(* CODESYS project cnc_v3.project
   Version: 0.0.0.0
   Title: cnc
   Author: Officina

Project tree, tasks and I/O mapping:
  MyController : TM241C24R, Schneider Electric, order no. TM241C24R, version 5.0.8.2
    application Application
      libraries: SysTimeCore, * (System); MemoryUtils, * (3S - Smart Software Solutions GmbH); CAA Mathematics, * (CAA Technical Workgroup); FloatingPointUtils, * (System); VisuDialogs, * (System)
      task MAST (cyclic, interval 20 ms, priority 15, watchdog 100 ms x 1) calls test
      program test [CFC]
      cnc/
        function block cnc [ST]: line_lenght, sc_char_is_letter, sc_findp, sc_find_nonum, sc_find_num, sc_get_letter, sc_get_value, sc_parse_clean, sc_parse_line, sc_parse_start, to_upper, trim, uppercase, arc_lenght, line_arc_angle, arc_arc_angle, line_line_angle, arc_line_angle, p_to_v, get_blockangles, get_corner_ve_blockangles, sc_get_gforce, get_velmax_gforce, sc_optimize_all, sc_optimize_G0_ve, sc_optimize_G123_ve_backward, sc_optimize_G123_ve_forward, sc_set_gforce, interpolate_lenght, interpolate_arc, update_motion_and_interpolator, interpolate_line, round, netto, set_pnt_at
        structure/
          data type sc_motion_status
          data type sc_data
          data type sc_enum_program_status
          data type sc_segment
          data type coordinate_type
          data type sc_pnt
          data type sc_primitive_id
          data type ascii_letters
          data type sc_dir
          data type sc_ext
          data type cn_jog_cmd
          data type cn_limits
        vector3/
          function V3_ANG [ST]
          function V3_DOT [ST]
          function V3_NORMALIZED [ST]
          function V3_NUL [ST]
          function V3_PAR [ST]
          function V3_REV [ST]
          function V3_SMUL [ST]
          function V3_SUB [ST]
          function V3_XANG [ST]
          function V3_CROSS [ST]
          function V3_YANG [ST]
          function V3_ZANG [ST]
          function V3_COPY [ST]
          function V3_NORM [ST]
          function V3_SDIV [ST]
          data type Vector_3
          function V3_ABS [ST]
          function V3_ADD [ST]
        motion/
          function block sc_engine [ST]: set_data, get_result, set_cycle_time, update, motion, Sc_bck, Sc_fwd, get_status, set_pos, set_jog, jog_stop
        global variables CN_CONSTANT
        vector/
          functions/
            function vector_traject_lenght [ST]
            function vector_nr_decrement [ST]
            function vector_at [ST]
            function vector_nr_increment [ST]
            function round [ST]
          function block vector_sc_segment [ST]: clear, end, begin, push_back, back, front, size, insert
        global variables CN_SETTINGS
      trace Traccia (task MAST): test.x, test.y, test.z, test.velocity, test.acceleration
      visualisation Visualization
      new/
        function block sc_parser [ST]: arc_lenght, line_lenght, sc_char_is_letter, sc_findp, sc_find_nonum, sc_find_num, sc_get_letter, sc_get_value, sc_parse_clean, sc_parse_line, sc_parse_start, to_upper, trim, uppercase
        function block sc_optimizer [ST]: arc_arc_angle, arc_line_angle, get_blockangles, get_corner_ve_blockangles, get_velmax_gforce, line_arc_angle, line_line_angle, p_to_v, sc_get_gforce, sc_optimize_all, sc_optimize_G0_ve, sc_optimize_G123_ve_backward, sc_optimize_G123_ve_forward, sc_set_gforce
    Serial_Line_2 : Serial line, Schneider Electric, version 5.0.8.2
      Modbus_Manager : Modbus Manager, Schneider Electric, version 4.0.0.3
    DI : Digital Inputs, Schneider Electric, version 5.0.8.2
        input  iwDI_IW0 : WORD  // IW0
        input  ibDI_IB1 : BYTE  // IB1
    DQ : Digital Outputs, Schneider Electric, version 5.0.8.2
        output qwDQ_QW0 : WORD  // QW0
        output qbDQ_QB1 : BYTE  // QB1
    Counters : Counters, Schneider Electric, version 5.0.8.2
    Pulse_Generators : Pulse Generators, Schneider Electric, version 5.0.8.2
    IO_Bus : IO bus - TM3, Schneider Electric, version 5.0.8.2
    Serial_Line_1 : Serial line, Schneider Electric, version 5.0.8.2
      Machine_Expert_Network_Manager : Machine Expert-Network Manager, Schneider Electric, version 4.0.0.3
    Cartridge_1 : Cartridge, Schneider Electric, version 5.0.8.2
    COM_Bus : COM bus, Schneider Electric, version 5.0.8.2
  libraries: VisuSymbols, 3.5.10.0 (System)
  text list GlobalTextList
*)

// MyController/Application/cnc/structure/sc_motion_status
TYPE sc_motion_status :
(
	motion_error,
	motion_finish,
	motion_pause,
	motion_process
);
END_TYPE

// MyController/Application/cnc/structure/sc_data
TYPE sc_data :
STRUCT
	sc_ct:LREAL;//scurve curve time                 //
	sc_jm:LREAL;//jerk result                       //
 	sc_cs:LREAL;//curve displacement                //
	sc_vr:LREAL;//velocity resul                    //
	sc_sr:LREAL;//position result                   //  result
	sc_ar:LREAL;//acceleration result               //
	tr_ct:LREAL;//total curve time                  //
 	tr_cs:LREAL;//total curve displacement          //
	at_time:LREAL;//request at timestamp.			//
	cycle_time:LREAL;
	state:sc_motion_status;
	
	ds:LREAL;//target
	vo:LREAL;//begin velocity
	ve:LREAL;//end velocity
	vs:LREAL;//max velocity
	a:LREAL;//acceleration
	gain:LREAL;//0-100
	
	ds_old:LREAL;//target old
	vs_old:LREAL;//max velocity old
	sc_sr_inc:LREAL;//position result incremental
	sc_sr_inc_old:LREAL;//position result incremental old
		
	init:BOOL;//new move reinit
	stop:BOOL;
	zero_vel_acc:BOOL;
	
	dir:INT;//movement direction
	
	t_vin:LREAL;
	t_pos:LREAL;
	
	finish:BOOL;
	
	jog_stop:BOOL;
	jog_fwd:BOOL;
	jog_rev:BOOL;
	
END_STRUCT
END_TYPE

// MyController/Application/cnc/structure/sc_enum_program_status

TYPE sc_enum_program_status :
(
	program_start:=0,
	program_run:=1,
	program_pause:=2,
	program_pause_resume:=3,
	program_stop:=4,
	program_vm_interupt:=5,
	program_wait:=6,
	program_end:=7,
	program_jog:=8,
	program_error:=9
);
END_TYPE

// MyController/Application/cnc/structure/sc_segment
TYPE sc_segment :
STRUCT
	primitive_id:sc_primitive_id;
    gcode_line_nr:UDINT;
    pnt_s:sc_pnt; 
	pnt_e:sc_pnt;
	pnt_c:sc_pnt;
   	dir_s:sc_dir; 
	dir_e:sc_dir;
    ext_s:sc_ext; 
	ext_e:sc_ext;
	radius:LREAL;
    angle_end:LREAL;
	vel_start:LREAL;
	vel_max:LREAL;
    vel_end:LREAL;
	acc_start:LREAL;
	acc_end:LREAL;
    traject_lenght_begin:LREAL;
	traject_lenght_end:LREAL;
    path_lenght:LREAL;
	m_value:UDINT;
	s_value:UDINT;
	s_dir:BOOL; //! spindle direction (1cw -0ccw)
	p_value:UDINT;
	t_value:UDINT;
	h_value:UDINT;
	abs_inc:BOOL;//abs / inc coordinate 
	back_optim:BOOL;
	forward_optim:BOOL;
END_STRUCT
END_TYPE

// MyController/Application/cnc/structure/coordinate_type

TYPE coordinate_type :
(
	abs_coord := 0,
	inc_coord := 1
);
END_TYPE

// MyController/Application/cnc/structure/sc_pnt
TYPE sc_pnt :
STRUCT
	x,y,z:LREAL;
END_STRUCT
END_TYPE

// MyController/Application/cnc/structure/sc_primitive_id

TYPE sc_primitive_id :
(
	empty:=0,
	rapid:=1,
	line:=2,
	arc_cw:=3,
	arc_ccw:=4	
);
END_TYPE

// MyController/Application/cnc/structure/ascii_letters

TYPE ascii_letters :
(
        A_ := 65,
        B_ := 66,
        C_ := 67,
        D_ := 68,
        E_ := 69,
        F_ := 70,
        G_ := 71,
        H_ := 72,
        I_ := 73,
        J_ := 74,
        K_ := 75,
        L_ := 76,
        M_ := 77,
        N_ := 78,
        O_ := 79,
        P_ := 80,
        Q_ := 81,
        R_ := 82,
        S_ := 83,
        T_ := 84,
        U_ := 85,
        V_ := 86,
        W_ := 87,
        X_ := 88,
        Y_ := 89,
        Z_ := 90
);
END_TYPE

// MyController/Application/cnc/structure/sc_dir
TYPE sc_dir :
STRUCT
	a:LREAL;
	b:LREAL;
	c:LREAL;
END_STRUCT
END_TYPE

// MyController/Application/cnc/structure/sc_ext
TYPE sc_ext :
STRUCT
	u:LREAL;
	v:LREAL;
	w:LREAL;
END_STRUCT
END_TYPE

// MyController/Application/cnc/vector3/Vector_3
TYPE Vector_3 :
STRUCT
	x:LREAL;
	y:LREAL;
	z:LREAL;
END_STRUCT
END_TYPE

// MyController/Application/cnc/structure/cn_jog_cmd
TYPE cn_jog_cmd :
STRUCT
	jog_enable:BOOL;
	x_up:BOOL;
	x_dn:BOOL;
	y_up:BOOL;
	y_dn:BOOL;
	z_up:BOOL;
	z_dp:BOOL;
END_STRUCT
END_TYPE

// MyController/Application/cnc/structure/cn_limits
TYPE cn_limits :
STRUCT
	max_vel:LREAL;
	max_acc:LREAL;
	max_jerk:LREAL;
	max_quote_x:LREAL;
	min_quote_x:LREAL;
	max_quote_y:LREAL;
	min_quote_y:LREAL;
	max_quote_z:LREAL;
	min_quote_z:LREAL;
END_STRUCT
END_TYPE

// MyController/Application/cnc/CN_CONSTANT
VAR_GLOBAL CONSTANT	
	DECIMALS:INT:=3;
	INFINITY:LREAL:=3.402823E+38;			
	M_PI:LREAL:=3.14159265358979323846264338327950288;
	TO_DEGREES:LREAL:=180/M_PI;
END_VAR

// MyController/Application/cnc/CN_SETTINGS
VAR_GLOBAL CONSTANT
	ANGLE_VEL_FACTOR:LREAL:=1;// 0-1
	STOP_ANGLE:LREAL:=90; 
	CT:LREAL:=0.02; //cycle time
	MAX_LOOK_HEAD_LINE:UDINT:=50;
	MAX_GCODE_LINE:UDINT:=2500;
	MAX_TOOLS:UINT:=10;
END_VAR

// MyController/Application/test
PROGRAM test
VAR
	cnc_0: cnc;
	feed_override: LREAL:=100;
	adaptive_feed: LREAL:=100;
	maxacc: LREAL:=250;
	maxjerk: LREAL:=100;
	maxvel: LREAL:=250;
	start: BOOL;
	stop: BOOL;
	pause: BOOL;
	start_line: UDINT;
	x: LREAL;
	y: LREAL;
	z: LREAL;
	velocity: LREAL;
	acceleration: LREAL;
	traject_progress: LREAL;
	line_progress: LREAL;
	performance: LREAL;
	line_nr: UDINT;
	jog_enable: BOOL;
	gcode:ARRAY [0..MAX_GCODE_LINE]OF STRING (250)
	:=[		
		
'G1 X0 Y50 z0 F150 						',			
'G1 X10 Y100 z0							',
'G1 X0 Y150 z0 							',
'G2 X150 Y0 z-15 I0 J-150 				',
'G0 z2                          ',
'G00 X-25.967 Y-14.626 Z2.000   ',
'G00 X0.033 Y0.040 Z2.000       ',
'G01 X0.033 Y0.040 Z-0.160 F50 ',
'G01 X-0.078 Y-0.152 Z-0.160    ',
'G01 X-0.189 Y0.425 Z-0.242     ',
'G01 X0.700 Y0.040 Z-0.019      ',
'G01 X0.601 Y-0.436 Z-0.019     ',
'G01 X0.175 Y-0.762 Z-0.097     ',
'G01 X-0.411 Y-0.729 Z-0.343    ',
'G01 X-0.872 Y-0.289 Z-0.610    ',
'G01 X-0.941 Y0.395 Z-0.610     ',
'G01 X-0.522 Y1.003 Z-0.347     ',
'G01 X0.239 Y1.208 Z-0.102      ',
'G01 X0.998 Y0.850 Z-0.005      ',
'G01 X1.367 Y0.040 Z0.000       ',
'G01 X1.292 Y-0.520 Z0.000      ',
'G01 X0.985 Y-1.016 Z-0.006     ',
'G01 X0.487 Y-1.354 Z-0.058     ',
'G01 X-0.125 Y-1.462 Z-0.267    ',
'G01 X-0.744 Y-1.307 Z-0.486    ',
'G01 X-1.261 Y-0.900 Z-0.937    ',
'G01 X-1.575 Y-0.301 Z-1.036    ',
'G01 X-1.619 Y0.392 Z-1.036     ',
'G01 X-1.369 Y1.059 Z-0.951     ',
'G01 X-0.856 Y1.580 Z-0.660     ',
'G01 X-0.157 Y1.853 Z-0.288     ',
'G01 X0.610 Y1.816 Z-0.035      ',
'G01 X1.312 Y1.461 Z0.000       ',
'G01 X1.820 Y0.836 Z0.000       ',
'G01 X2.033 Y0.040 Z0.000       ',
'G01 X1.975 Y-0.558 Z0.000      ',
'G01 X1.738 Y-1.122 Z0.000      ',
'G01 X1.340 Y-1.598 Z0.000      ',
'G01 X0.810 Y-1.939 Z-0.038     ',
'G01 X0.195 Y-2.112 Z-0.151     ',
'G01 X-0.454 Y-2.095 Z-0.437    ',
'G01 X-1.078 Y-1.884 Z-0.881    ',
'G01 X-1.619 Y-1.493 Z-1.085    ',
'G01 X-2.026 Y-0.951 Z-1.114    ',
'G01 X-2.258 Y-0.305 Z-1.114    ',
'G01 X-2.290 Y0.391 Z-1.114     ',
'G01 X-2.112 Y1.074 Z-1.117     ',
'G01 X-1.735 Y1.682 Z-1.134     ',
'G01 X-1.189 Y2.157 Z-0.927     ',
'G01 X-0.518 Y2.455 Z-0.478     ',
'G01 X0.221 Y2.541 Z-0.174      ',
'G01 X0.961 Y2.405 Z-0.028      ',
'G01 X1.637 Y2.051 Z0.000       ',
'G01 X2.184 Y1.507 Z0.000       ',
'G01 X2.551 Y0.817 Z0.000       ',
'G01 X2.700 Y0.040 Z0.000       ',
'G01 X2.656 Y-0.558 Z0.000      ',
'G01 X2.479 Y-1.137 Z0.000      ',
'G01 X2.174 Y-1.667 Z0.000      ',
'G01 X1.755 Y-2.119 Z0.000      ',
'G01 X1.242 Y-2.469 Z-0.007     ',
'G01 X0.659 Y-2.699 Z-0.071     ',
'G01 X0.033 Y-2.793 Z-0.303     ',
'G01 X-0.602 Y-2.745 Z-0.691    ',
'G01 X-1.217 Y-2.555 Z-1.150    ',
'G01 X-1.778 Y-2.231 Z-1.189    ',
'G01 X-2.256 Y-1.785 Z-1.144    ',
'G01 X-2.627 Y-1.241 Z-1.131    ',
'G01 X-2.868 Y-0.622 Z-1.120    ',
'G01 X-2.967 Y0.040 Z-1.119     ',
'G01 X-2.915 Y0.713 Z-1.120     ',
'G01 X-2.712 Y1.363 Z-1.134     ',
'G01 X-2.368 Y1.955 Z-1.175     ',
'G01 X-1.897 Y2.460 Z-1.230     ',
'G01 X-1.320 Y2.851 Z-1.221     ',
'G01 X-0.666 Y3.105 Z-0.765     ',
'G01 X0.033 Y3.207 Z-0.352      ',
'G01 X0.743 Y3.151 Z-0.112      ',
'G01 X1.428 Y2.936 Z-0.006      ',
'G01 X2.052 Y2.572 Z0.000       ',
'G01 X2.584 Y2.074 Z0.000       ',
'G00 X120 Y120 Z0.000       ',
'G01 X2.994 Y1.466 Z0.000       ',
'G01 X3.260 Y0.777 Z-0.008      ',
'G01 X3.367 Y0.040 Z-0.015      ',
'G01 X3.329 Y-0.576 Z-0.009     ',
'G01 X3.178 Y-1.178 Z0.000      ',
'G01 X2.917 Y-1.745 Z0.000      ',
'G01 X2.555 Y-2.258 Z0.000      ',
'G01 X2.101 Y-2.698 Z0.000      ',
'G01 X1.572 Y-3.049 Z0.000      ',
'G01 X0.983 Y-3.298 Z-0.077     ',
'G01 X0.355 Y-3.435 Z-0.317     ',
'G01 X-0.291 Y-3.454 Z-0.548    ',
'G01 X-0.933 Y-3.354 Z-0.977    ',
'G01 X-1.549 Y-3.136 Z-1.340    ',
'G01 X-2.117 Y-2.807 Z-1.291    ',
'G01 X-2.618 Y-2.377 Z-1.228    ',
'G01 X-3.034 Y-1.859 Z-1.205    ',
'G01 X-3.349 Y-1.270 Z-1.167    ',
'G01 X-3.552 Y-0.630 Z-1.156    ',
'G01 X-3.633 Y0.040 Z-1.156     ',
'G01 X-3.590 Y0.718 Z-1.157     ',
'G01 X-3.422 Y1.379 Z-1.193     ',
'G01 X-3.134 Y2.002 Z-1.212     ',
'G01 X-2.734 Y2.564 Z-1.241     ',
'G01 X-2.235 Y3.045 Z-1.357     ',
'G01 X-1.653 Y3.428 Z-1.410     ',
'G01 X-1.008 Y3.699 Z-1.251     ',
'G01 X-0.319 Y3.848 Z-0.791     ',
'G01 X0.388 Y3.867 Z-0.280      ',
'G01 X1.090 Y3.756 Z-0.084      ',
'G01 X1.764 Y3.516 Z-0.001      ',
'G01 X2.385 Y3.154 Z0.000       ',
'G01 X2.931 Y2.682 Z0.000       ',
'G01 X3.384 Y2.115 Z0.000       ',
'G01 X3.727 Y1.471 Z-0.032      ',
'G01 X3.946 Y0.772 Z-0.114      ',
'G01 X4.033 Y0.040 Z-0.149      ',
'G01 X4.001 Y-0.588 Z-0.119     ',
'G01 X3.869 Y-1.206 Z-0.036     ',
'G01 X3.642 Y-1.798 Z-0.004     ',
'G01 X3.323 Y-2.350 Z0.000      ',
'G01 X2.921 Y-2.847 Z0.000      ',
'G01 X2.443 Y-3.277 Z0.000      ',
'G01 X1.902 Y-3.628 Z-0.004     ',
'G01 X1.311 Y-3.891 Z-0.058     ',
'G01 X0.683 Y-4.058 Z-0.226     ',
'G01 X0.033 Y-4.126 Z-0.603     ',
'G01 X-0.621 Y-4.091 Z-1.092    ',
'G01 X-1.265 Y-3.954 Z-1.537    ',
'G01 X-1.881 Y-3.717 Z-1.507    ',
'G01 X-2.455 Y-3.384 Z-1.391    ',
'G01 X-2.972 Y-2.965 Z-1.381    ',
'G01 X-3.418 Y-2.467 Z-1.313    ',
'G01 X-3.783 Y-1.904 Z-1.281    ',
'G01 X-4.056 Y-1.288 Z-1.238    ',
'G01 X-4.230 Y-0.635 Z-1.244    ',
'G01 X-4.300 Y0.040 Z-1.244     ',
'G01 X-4.263 Y0.721 Z-1.245     ',
'G01 X-4.120 Y1.390 Z-1.278     ',
'G01 X-3.872 Y2.030 Z-1.325     ',
'G01 X-3.526 Y2.627 Z-1.362     ',
'G01 X-3.090 Y3.164 Z-1.399     ',
'G01 X-2.573 Y3.627 Z-1.480     ',
'G01 X-1.987 Y4.005 Z-1.604     ',
'G01 X-1.347 Y4.289 Z-1.652     ',
'G01 X-0.668 Y4.469 Z-1.209     ',
'G01 X0.033 Y4.540 Z-0.707      ',
'G01 X0.740 Y4.502 Z-0.343      ',
'G01 X1.434 Y4.352 Z-0.092      ',
'G01 X2.099 Y4.095 Z-0.003      ',
'G01 X2.718 Y3.735 Z0.000       ',
'G01 X3.274 Y3.281 Z0.000       ',
'G01 X3.755 Y2.744 Z0.000       ',
'G01 X4.147 Y2.136 Z-0.052      ',
'G01 X4.440 Y1.472 Z-0.178      ',
'G01 X4.626 Y0.768 Z-0.364      ',
'G01 X4.700 Y0.040 Z-0.441      ',
'G01 X4.672 Y-0.583 Z-0.375     ',
'G01 X4.562 Y-1.200 Z-0.190     ',
'G01 X4.369 Y-1.798 Z-0.132     ',
'G01 X4.097 Y-2.367 Z-0.008     ',
'G01 X3.751 Y-2.896 Z0.000      ',
'G01 X3.337 Y-3.375 Z0.000      ',
'G01 X2.860 Y-3.796 Z0.000      ',
'G01 X2.331 Y-4.151 Z0.000      ',
'G01 X1.756 Y-4.434 Z-0.037     ',
'G01 X1.148 Y-4.637 Z-0.213     ',
'G01 X0.516 Y-4.758 Z-0.566     ',
'G01 X-0.128 Y-4.794 Z-1.019    ',
'G01 X-0.774 Y-4.743 Z-1.551    ',
'G01 X-1.408 Y-4.606 Z-1.798    ',
'G01 X-2.021 Y-4.386 Z-1.732    ',
'G01 X-2.600 Y-4.084 Z-1.662    ',
'G01 X-3.135 Y-3.707 Z-1.554    ',
'G01 X-3.617 Y-3.261 Z-1.486    ',
'G01 X-4.036 Y-2.753 Z-1.464    ',
'G01 X-4.385 Y-2.192 Z-1.422    ',
'G01 X-4.657 Y-1.588 Z-1.375    ',
'G01 X-4.846 Y-0.951 Z-1.380    ',
'G01 X-4.948 Y-0.293 Z-1.376    ',
'G01 X-4.963 Y0.375 Z-1.376     ',
'G01 X-4.887 Y1.041 Z-1.394     ',
'G01 X-4.724 Y1.692 Z-1.382     ',
'G01 X-4.474 Y2.318 Z-1.437     ',
'G01 X-4.141 Y2.906 Z-1.524     ',
'G01 X-3.733 Y3.447 Z-1.542     ',
'G01 X-3.254 Y3.929 Z-1.602     ',
'G01 X-2.714 Y4.345 Z-1.692     ',
'G01 X-2.122 Y4.685 Z-1.851     ',
'G01 X-1.488 Y4.945 Z-1.946     ',
'G01 X-0.823 Y5.118 Z-1.696     ',
'G01 X-0.139 Y5.201 Z-1.159     ',
'G01 X0.552 Y5.192 Z-0.687      ',
'G01 X1.237 Y5.091 Z-0.349      ',
'G01 X1.904 Y4.898 Z-0.099      ',
'G01 X2.542 Y4.618 Z-0.006      ',
'G01 X3.138 Y4.254 Z0.000       ',
'G01 X3.682 Y3.813 Z0.000       ',
'G01 X4.163 Y3.302 Z0.000       ',
'G01 X4.573 Y2.729 Z-0.029      ',
'G01 X4.904 Y2.106 Z-0.213      ',
'G01 X5.150 Y1.442 Z-0.464      ',
'G01 X5.305 Y0.749 Z-0.798      ',
'G01 X5.367 Y0.040 Z-0.948      ',
'G01 X5.342 Y-0.592 Z-0.819     ',
'G01 X5.242 Y-1.218 Z-0.485     ',
'G01 X5.068 Y-1.830 Z-0.367     ',
'G01 X4.823 Y-2.418 Z-0.144     ',
'G01 X4.509 Y-2.974 Z-0.008     ',
'G01 X4.131 Y-3.491 Z0.000      ',
'G01 X3.693 Y-3.960 Z0.000      ',
'G01 X3.201 Y-4.375 Z0.000      ',
'G01 X2.663 Y-4.729 Z0.000      ',
'G01 X2.085 Y-5.018 Z-0.083     ',
'G01 X1.476 Y-5.238 Z-0.307     ',
'G01 X0.843 Y-5.384 Z-0.496     ',
'G01 X0.196 Y-5.454 Z-1.012     ',
'G01 X-0.456 Y-5.447 Z-1.513    ',
'G01 X-1.104 Y-5.363 Z-1.966    ',
'G01 X-1.739 Y-5.203 Z-2.116    ',
'G01 X-2.352 Y-4.968 Z-2.012    ',
'G01 X-2.935 Y-4.661 Z-1.843    ',
'G01 X-3.478 Y-4.287 Z-1.752    ',
'G01 X-3.974 Y-3.850 Z-1.753    ',
'G01 X-4.416 Y-3.356 Z-1.657    ',
'G01 X-4.797 Y-2.812 Z-1.657    ',
'G01 X-5.112 Y-2.226 Z-1.574    ',
'G01 X-5.356 Y-1.605 Z-1.542    ',
'G01 X-5.525 Y-0.959 Z-1.565    ',
'G01 X-5.617 Y-0.295 Z-1.560    ',
'G01 X-5.630 Y0.377 Z-1.560     ',
'G01 X-5.563 Y1.046 Z-1.579     ',
'G01 X-5.416 Y1.705 Z-1.618     ',
'G01 X-5.193 Y2.343 Z-1.648     ',
'G01 X-4.895 Y2.951 Z-1.679     ',
'G01 X-4.526 Y3.521 Z-1.796     ',
'G01 X-4.091 Y4.045 Z-1.825     ',
'G01 X-3.597 Y4.514 Z-1.863     ',
'G01 X-3.049 Y4.923 Z-1.990     ',
'G01 X-2.455 Y5.264 Z-2.159     ',
'G01 X-1.824 Y5.534 Z-2.272     ',
'G01 X-1.164 Y5.727 Z-2.270     ',
'G01 X-0.484 Y5.841 Z-1.679     ',
'G01 X0.206 Y5.874 Z-1.173      ',
'G01 X0.897 Y5.825 Z-0.732      ',
'G01 X1.578 Y5.695 Z-0.322      ',
'G01 X2.241 Y5.484 Z-0.093      ',
'G01 X2.875 Y5.196 Z-0.006      ',
'G01 X3.473 Y4.834 Z0.000       ',
'G01 X4.024 Y4.402 Z0.000       ',
'G01 X4.521 Y3.908 Z0.000       ',
'G01 X4.958 Y3.357 Z-0.017      ',
'G01 X5.327 Y2.757 Z-0.197      ',
'G01 X5.622 Y2.117 Z-0.485      ',
'G01 X5.841 Y1.444 Z-0.916      ',
'G01 X5.979 Y0.749 Z-1.420      ',
'G01 X6.033 Y0.040 Z-1.593      ',
'G01 X6.011 Y-0.599 Z-1.449     ',
'G01 X5.920 Y-1.233 Z-0.955     ',
'G01 X5.762 Y-1.855 Z-0.637     ',
'G01 X5.538 Y-2.457 Z-0.357     ',
'G01 X5.251 Y-3.034 Z-0.077     ',
'G01 X4.904 Y-3.578 Z-0.009     ',
'G01 X4.500 Y-4.083 Z0.000      ',
'G01 X4.044 Y-4.543 Z0.000      ',
'G01 X3.541 Y-4.953 Z0.000      ',
'G01 X2.995 Y-5.307 Z-0.010     ',
'G01 X2.415 Y-5.602 Z-0.081     ',
'G01 X1.805 Y-5.834 Z-0.291     ',
'G01 X1.172 Y-6.000 Z-0.672     ',
'G01 X0.525 Y-6.098 Z-1.221     ',
'G01 X-0.131 Y-6.127 Z-1.716    ',
'G01 X-0.787 Y-6.086 Z-2.294    ',
'G01 X-1.436 Y-5.975 Z-2.477    ',
'G01 X-2.071 Y-5.795 Z-2.349    ',
'G01 X-2.684 Y-5.548 Z-2.241    ',
'G01 X-3.269 Y-5.238 Z-2.187    ',
'G01 X-3.818 Y-4.865 Z-2.050    ',
'G01 X-4.326 Y-4.436 Z-2.009    ',
'G01 X-4.786 Y-3.955 Z-1.973    ',
'G01 X-5.193 Y-3.426 Z-1.972    ',
'G01 X-5.541 Y-2.856 Z-1.847    ',
'G01 X-5.828 Y-2.251 Z-1.776    ',
'G01 X-6.050 Y-1.618 Z-1.761    ',
'G01 X-6.203 Y-0.964 Z-1.808    ',
'G01 X-6.285 Y-0.296 Z-1.794    ',
'G01 X-6.297 Y0.378 Z-1.794     ',
'G01 X-6.236 Y1.051 Z-1.813     ',
'G01 X-6.104 Y1.714 Z-1.884     ',
'G01 X-5.902 Y2.361 Z-1.872     ',
'G01 X-5.632 Y2.984 Z-1.869     ',
'G01 X-5.296 Y3.576 Z-1.996     ',
'G01 X-4.899 Y4.130 Z-2.000     ',
'G01 X-4.444 Y4.639 Z-2.134     ',
'G01 X-3.937 Y5.097 Z-2.232     ',
'G01 X-3.383 Y5.500 Z-2.346     ',
'G01 X-2.788 Y5.843 Z-2.420     ',
'G01 X-2.159 Y6.120 Z-2.527     ',
'G01 X-1.503 Y6.330 Z-2.662     ',
'G01 X-0.828 Y6.469 Z-2.500     ',
'G01 X-0.140 Y6.535 Z-1.913     ',
'G01 X0.553 Y6.528 Z-1.407      ',
'G01 X1.241 Y6.447 Z-0.970      ',
'G01 X1.919 Y6.293 Z-0.490      ',
'G01 X2.577 Y6.068 Z-0.186      ',
'G01 X3.209 Y5.773 Z-0.035      ',
'G01 X3.807 Y5.413 Z0.000       ',
'G01 X4.364 Y4.990 Z0.000       ',
'G01 X4.874 Y4.509 Z0.000       ',
'G01 X5.330 Y3.976 Z-0.002      ',
'G01 X5.728 Y3.396 Z-0.115      ',
'G01 X6.063 Y2.777 Z-0.382      ',
'G01 X6.330 Y2.124 Z-0.855      ',
'G01 X6.527 Y1.445 Z-1.478      ',
'G01 X6.651 Y0.748 Z-1.901      ',
'G01 X6.700 Y0.040 Z-2.052      ',
'G01 X6.679 Y-0.604 Z-1.927     ',
'G01 X6.596 Y-1.244 Z-1.670     ',
'G01 X6.451 Y-1.875 Z-1.055     ',
'G01 X6.246 Y-2.489 Z-0.620     ',
'G01 X5.982 Y-3.082 Z-0.243     ',
'G01 X5.661 Y-3.647 Z-0.030     ',
'G01 X5.287 Y-4.179 Z0.000      ',
'G01 X4.863 Y-4.674 Z0.000      ',
'G01 X4.392 Y-5.126 Z0.000      ',
'G01 X3.879 Y-5.531 Z0.000      ',
'G01 X3.328 Y-5.885 Z-0.030     ',
'G01 X2.745 Y-6.184 Z-0.168     ',
'G01 X2.135 Y-6.427 Z-0.456     ',
'G01 X1.503 Y-6.609 Z-0.792     ',
'G01 X0.855 Y-6.730 Z-1.198     ',
'G01 X0.198 Y-6.788 Z-1.810     ',
'G01 X-0.462 Y-6.783 Z-2.357    ',
'G01 X-1.120 Y-6.713 Z-2.815    ',
'G01 X-1.769 Y-6.580 Z-2.908    ',
'G01 X-2.403 Y-6.385 Z-2.762    ',
'G01 X-3.017 Y-6.129 Z-2.660    ',
'G01 X-3.603 Y-5.814 Z-2.456    ',
'G01 X-4.158 Y-5.444 Z-2.467    ',
'G01 X-4.674 Y-5.022 Z-2.359    ',
'G01 X-5.149 Y-4.550 Z-2.299    ',
'G01 X-5.576 Y-4.035 Z-2.198    ',
'G01 X-5.952 Y-3.480 Z-2.202    ',
'G01 X-6.273 Y-2.890 Z-2.091    ',
'G01 X-6.536 Y-2.271 Z-2.134    ',
'G01 X-6.738 Y-1.629 Z-2.063    ',
'G01 X-6.878 Y-0.969 Z-2.104    ',
'G01 X-6.953 Y-0.297 Z-2.088    ',
'G01 X-6.964 Y0.379 Z-2.088     ',
'G01 X-6.908 Y1.054 Z-2.109     ',
'G01 X-6.788 Y1.722 Z-2.178     ',
'G01 X-6.604 Y2.376 Z-2.194     ',
'G01 X-6.357 Y3.010 Z-2.205     ',
'G01 X-6.049 Y3.618 Z-2.232     ',
'G01 X-5.684 Y4.194 Z-2.401     ',
'G01 X-5.264 Y4.733 Z-2.410     ',
'G01 X-4.793 Y5.230 Z-2.466     ',
'G01 X-4.276 Y5.680 Z-2.513     ',
'G01 X-3.717 Y6.078 Z-2.674     ',
'G01 X-3.121 Y6.421 Z-2.863     ',
'G01 X-2.494 Y6.705 Z-2.972     ',
'G01 X-1.842 Y6.928 Z-3.134     ',
'G01 X-1.170 Y7.087 Z-3.209     ',
'G01 X-0.485 Y7.181 Z-2.591     ',
'G01 X0.207 Y7.208 Z-2.028      ',
'G01 X0.899 Y7.168 Z-1.544      ',
'G01 X1.585 Y7.061 Z-1.110      ',
'G01 X2.258 Y6.888 Z-0.604      ',
'G01 X2.913 Y6.651 Z-0.264      ',
'G01 X3.542 Y6.351 Z-0.042      ',
'G01 X4.141 Y5.991 Z-0.003      ',
'G01 X4.703 Y5.575 Z0.000       ',
'G01 X5.222 Y5.106 Z0.000       ',
'G01 X5.695 Y4.588 Z0.000       ',
'G01 X6.116 Y4.025 Z-0.026      ',
'G01 X6.481 Y3.425 Z-0.225      ',
'G01 X6.787 Y2.790 Z-0.601      ',
'G01 X7.031 Y2.129 Z-1.240      ',
'G01 X7.210 Y1.445 Z-1.833      ',
'G01 X7.322 Y0.747 Z-2.229      ',
'G01 X7.367 Y0.040 Z-2.370      ',
'G01 X7.348 Y-0.599 Z-2.253     ',
'G01 X7.273 Y-1.236 Z-1.957     ',
'G01 X7.144 Y-1.865 Z-1.415     ',
'G01 X6.959 Y-2.480 Z-0.908     ',
'G01 X6.722 Y-3.078 Z-0.396     ',
'G01 X6.432 Y-3.654 Z-0.116     ',
'G01 X6.094 Y-4.203 Z-0.011     ',
'G01 X5.708 Y-4.721 Z0.000      ',
'G01 X5.278 Y-5.204 Z0.000      ',
'G01 X4.807 Y-5.648 Z0.000      ',
'G01 X4.298 Y-6.050 Z0.000      ',
'G01 X3.756 Y-6.407 Z-0.040     ',
'G01 X3.183 Y-6.715 Z-0.185     ',
'G01 X2.586 Y-6.972 Z-0.577     ',
'G01 X1.967 Y-7.177 Z-0.799     ',
'G01 X1.332 Y-7.327 Z-1.339     ',
'G01 X0.686 Y-7.422 Z-1.965     ',
'G01 X0.033 Y-7.460 Z-2.495     ',
'G01 X-0.621 Y-7.440 Z-3.113    ',
'G01 X-1.272 Y-7.364 Z-3.405    ',
'G01 X-1.915 Y-7.231 Z-3.428    ',
'G01 X-2.544 Y-7.042 Z-3.260    ',
'G01 X-3.156 Y-6.799 Z-3.127    ',
'G01 X-3.744 Y-6.503 Z-2.909    ',
'G01 X-4.306 Y-6.156 Z-2.921    ',
'G01 X-4.835 Y-5.762 Z-2.784    ',
'G01 X-5.329 Y-5.322 Z-2.695    ',
'G01 X-5.783 Y-4.840 Z-2.653    ',
'G01 X-6.194 Y-4.320 Z-2.652    ',
'G01 X-6.558 Y-3.765 Z-2.576    ',
'G01 X-6.873 Y-3.180 Z-2.457    ',
'G01 X-7.136 Y-2.569 Z-2.450    ',
'G01 X-7.345 Y-1.937 Z-2.432    ',
'G01 X-7.499 Y-1.288 Z-2.476    ',
'G01 X-7.595 Y-0.627 Z-2.443    ',
'G01 X-7.633 Y0.040 Z-2.442     ',
'G01 X-7.613 Y0.709 Z-2.444     ',
'G01 X-7.535 Y1.375 Z-2.484     ',
'G01 X-7.399 Y2.032 Z-2.447     ',
'G01 X-7.206 Y2.675 Z-2.593     ',
'G01 X-6.957 Y3.300 Z-2.555     ',
'G01 X-6.654 Y3.902 Z-2.607     ',
'G01 X-6.300 Y4.475 Z-2.689     ',
'G01 X-5.896 Y5.016 Z-2.796     ',
'G01 X-5.447 Y5.521 Z-2.953     ',
'G01 X-4.954 Y5.984 Z-2.970     ',
'G01 X-4.423 Y6.404 Z-3.130     ',
'G01 X-3.856 Y6.776 Z-3.127     ',
'G01 X-3.258 Y7.098 Z-3.396     ',
'G01 X-2.633 Y7.367 Z-3.512     ',
'G01 X-1.987 Y7.580 Z-3.698     ',
'G01 X-1.324 Y7.737 Z-3.885     ',
'G01 X-0.649 Y7.835 Z-3.394     ',
'G01 X0.033 Y7.874 Z-2.760      ',
'G01 X0.717 Y7.853 Z-2.200      ',
'G01 X1.397 Y7.773 Z-1.708      ',
'G01 X2.068 Y7.634 Z-1.138      ',
'G01 X2.725 Y7.436 Z-0.648      ',
'G01 X3.363 Y7.182 Z-0.306      ',
'G01 X3.978 Y6.872 Z-0.108      ',
'G01 X4.564 Y6.510 Z-0.009      ',
'G01 X5.116 Y6.098 Z0.000       ',
'G01 X5.631 Y5.638 Z0.000       ',
'G01 X6.105 Y5.135 Z0.000       ',
'G01 X6.533 Y4.592 Z-0.007      ',
'G01 X6.913 Y4.013 Z-0.087      ',
'G01 X7.242 Y3.402 Z-0.340      ',
'G01 X7.516 Y2.764 Z-0.871      ',
'G01 X7.734 Y2.104 Z-0.871      ',
'G01 X7.734 Y2.104 Z-1.566      ',
'G01 X7.894 Y1.426 Z-2.026      ',
'G01 X7.994 Y0.737 Z-2.378      ',
'G01 X8.033 Y0.040 Z-2.575      ',
'G01 X8.016 Y-0.604 Z-2.406     ',
'G01 X7.947 Y-1.246 Z-2.111     ',
'G01 X7.826 Y-1.880 Z-1.632     ',
'G01 X7.654 Y-2.504 Z-1.172     ',
'G01 X7.432 Y-3.112 Z-0.545     ',
'G01 X7.162 Y-3.701 Z-0.192     ',
'G01 X6.845 Y-4.267 Z-0.059     ',
'G01 X6.484 Y-4.807 Z0.000      ',
'G01 X6.079 Y-5.316 Z0.000      ',
'G01 X5.634 Y-5.791 Z0.000      ',
'G01 X5.152 Y-6.229 Z0.000      ',
'G01 X4.636 Y-6.628 Z-0.010     ',
'G01 X4.089 Y-6.984 Z-0.144     ',
'G01 X3.514 Y-7.295 Z-0.305     ',
'G01 X2.916 Y-7.560 Z-0.635     ',
'G01 X2.297 Y-7.775 Z-1.112     ',
'G01 X1.663 Y-7.940 Z-1.667     ',
'G01 X1.016 Y-8.054 Z-2.140     ',
'G01 X0.362 Y-8.115 Z-2.140     ',
'G01 X0.362 Y-8.115 Z-2.883     ',
'G01 X-0.296 Y-8.124 Z-3.305    ',
'G01 X-0.953 Y-8.079 Z-3.305    ',
'G01 X-0.953 Y-8.079 Z-4.019    ',
'G01 X-1.604 Y-7.982 Z-4.052    ',
'G01 X-2.247 Y-7.833 Z-3.830    ',
'G01 X-2.876 Y-7.631 Z-3.865    ',
'G01 X-3.488 Y-7.380 Z-3.553    ',
'G01 X-4.078 Y-7.080 Z-3.459    ',
'G01 X-4.642 Y-6.733 Z-3.302    ',
'G01 X-5.178 Y-6.342 Z-3.298    ',
'G01 X-5.680 Y-5.908 Z-3.278    ',
'G01 X-6.147 Y-5.435 Z-3.221    ',
'G01 X-6.574 Y-4.925 Z-3.093    ',
'G01 X-6.959 Y-4.381 Z-2.981    ',
'G01 X-7.300 Y-3.808 Z-2.933    ',
'G01 X-7.594 Y-3.209 Z-2.901    ',
'G01 X-7.839 Y-2.588 Z-2.841    ',
'G01 X-8.033 Y-1.948 Z-2.842    ',
'G01 X-8.175 Y-1.294 Z-2.903    ',
'G01 X-8.264 Y-0.629 Z-2.870    ',
'G01 X-8.300 Y0.040 Z-2.869     ',
'G01 X-8.281 Y0.712 Z-2.872     ',
'G01 X-8.209 Y1.380 Z-2.910     ',
'G01 X-8.083 Y2.041 Z-3.011     ',
'G01 X-7.904 Y2.690 Z-3.010     ',
'G01 X-7.672 Y3.324 Z-3.075     ',
'G01 X-7.391 Y3.937 Z-3.065     ',
'G01 X-7.060 Y4.526 Z-3.144     ',
'G01 X-6.683 Y5.088 Z-3.261     ',
'G01 X-6.262 Y5.617 Z-3.271     ',
'G01 X-5.799 Y6.112 Z-3.332     ',
'G01 X-5.297 Y6.568 Z-3.444     ',
'G01 X-4.759 Y6.983 Z-3.617     ',
'G01 X-4.189 Y7.354 Z-3.779     ',
'G01 X-3.590 Y7.677 Z-3.825     ',
'G01 X-2.967 Y7.952 Z-4.197     ',
'G01 X-2.323 Y8.176 Z-4.382     ',
'G01 X-1.663 Y8.348 Z-4.378     ',
'G01 X-0.990 Y8.466 Z-4.513     ',
'G01 X-0.309 Y8.529 Z-3.857     ',
'G01 X-0.309 Y8.529 Z-2.966     ',
'G01 X0.376 Y8.538 Z-2.966      ',
'G01 X1.059 Y8.491 Z-2.412      ',
'G01 X1.738 Y8.390 Z-1.945      ',
'G01 X2.407 Y8.234 Z-1.374      ',
'G01 X3.061 Y8.024 Z-0.885      ',
'G01 X3.697 Y7.762 Z-0.560      ',
'G01 X4.311 Y7.450 Z-0.197      ',
'G01 X4.898 Y7.089 Z-0.063      ',
'G01 X5.455 Y6.681 Z-0.002      ',
'G01 X5.978 Y6.229 Z0.000       ',
'G01 X6.463 Y5.737 Z0.000       ',
'G01 X6.907 Y5.206 Z0.000       ',
'G01 X7.308 Y4.641 Z-0.009      ',
'G01 X7.662 Y4.044 Z-0.135      ',
'G01 X7.967 Y3.421 Z-0.454      ',
'G01 X8.222 Y2.774 Z-0.954      ',
'G01 X8.423 Y2.108 Z-1.545      ',
'G01 X8.571 Y1.428 Z-2.007      ',
'G01 X8.663 Y0.737 Z-2.273      ',
'G01 X8.700 Y0.040 Z-2.419      ',
'G01 X8.684 Y-0.608 Z-2.302     ',
'G01 X8.619 Y-1.254 Z-1.996     ',
'G01 X8.506 Y-1.893 Z-1.610     ',
'G01 X8.345 Y-2.523 Z-1.034     ',
'G01 X8.138 Y-3.140 Z-0.654     ',
'G01 X7.885 Y-3.741 Z-0.254     ',
'G01 X7.587 Y-4.321 Z-0.050     ',
'G01 X7.247 Y-4.877 Z-0.001     ',
'G01 X6.865 Y-5.408 Z0.000      ',
'G01 X6.445 Y-5.908 Z0.000      ',
'G01 X5.988 Y-6.377 Z0.000      ',
'G01 X5.496 Y-6.810 Z-0.004     ',
'G01 X4.974 Y-7.206 Z-0.090     ',
'G01 X4.422 Y-7.561 Z-0.207     ',
'G01 X3.845 Y-7.875 Z-0.569     ',
'G01 X3.246 Y-8.145 Z-0.987     ',
'G01 X2.628 Y-8.370 Z-1.367     ',
'G01 X1.994 Y-8.548 Z-1.927     ',
'G01 X1.348 Y-8.679 Z-2.375     ',
'G01 X0.693 Y-8.760 Z-2.375     ',
'G01 X0.693 Y-8.760 Z-3.127     ',
'G01 X0.033 Y-8.793 Z-3.771     ',
'G01 X-0.627 Y-8.776 Z-3.771    ',
'G01 X-0.627 Y-8.776 Z-4.551    ',
'G01 X-1.286 Y-8.710 Z-4.783    ',
'G01 X-1.938 Y-8.595 Z-4.809    ',
'G01 X-2.580 Y-8.431 Z-4.559    ',
'G01 X-3.208 Y-8.219 Z-4.387    ',
'G01 X-3.820 Y-7.961 Z-4.237    ',
'G01 X-4.411 Y-7.658 Z-4.197    ',
'G01 X-4.978 Y-7.310 Z-4.023    ',
'G01 X-5.519 Y-6.922 Z-3.830    ',
'G01 X-6.029 Y-6.493 Z-3.702    ',
'G01 X-6.506 Y-6.027 Z-3.630    ',
'G01 X-6.947 Y-5.526 Z-3.613    ',
'G01 X-7.350 Y-4.994 Z-3.613    ',
'G01 X-7.713 Y-4.432 Z-3.529    ',
'G01 X-8.032 Y-3.844 Z-3.370    ',
'G01 X-8.308 Y-3.233 Z-3.526    ',
'G01 X-8.536 Y-2.603 Z-3.484    ',
'G01 X-8.718 Y-1.957 Z-3.332    ',
'G01 X-8.850 Y-1.299 Z-3.418    ',
'G01 X-8.934 Y-0.632 Z-3.382    ',
'G01 X-8.967 Y0.040 Z-3.381     ',
'G01 X-8.949 Y0.714 Z-3.384     ',
'G01 X-8.882 Y1.384 Z-3.426     ',
'G01 X-8.764 Y2.048 Z-3.529     ',
'G01 X-8.597 Y2.703 Z-3.508     ',
'G01 X-8.381 Y3.343 Z-3.558     ',
'G01 X-8.118 Y3.966 Z-3.675     ',
'G01 X-7.809 Y4.568 Z-3.573     ',
'G01 X-7.455 Y5.146 Z-3.813     ',
'G01 X-7.059 Y5.696 Z-3.810     ',
'G01 X-6.622 Y6.216 Z-3.989     ',
'G01 X-6.148 Y6.702 Z-4.069     ',
'G01 X-5.637 Y7.151 Z-4.213     ',
'G01 X-5.095 Y7.562 Z-4.316     ',
'G01 X-4.522 Y7.931 Z-4.520     ',
'G01 X-3.923 Y8.256 Z-4.633     ',
'G01 X-3.301 Y8.537 Z-4.741     ',
'G01 X-2.659 Y8.770 Z-4.935     ',
'G01 X-2.001 Y8.954 Z-5.214     ',
'G01 X-1.331 Y9.089 Z-5.512     ',
'G01 X-0.651 Y9.174 Z-4.953     ',
'G01 X-0.651 Y9.174 Z-4.123     ',
'G01 X0.033 Y9.207 Z-4.123      ',
'G01 X0.719 Y9.189 Z-3.445      ',
'G01 X1.402 Y9.120 Z-2.876      ',
'G01 X2.078 Y9.001 Z-2.195      ',
'G01 X2.745 Y8.830 Z-1.805      ',
'G01 X3.397 Y8.610 Z-1.290      ',
'G01 X4.031 Y8.342 Z-0.691      ',
'G01 X4.644 Y8.027 Z-0.383      ',
'G01 X5.233 Y7.667 Z-0.146      ',
'G01 X5.793 Y7.263 Z-0.046      ',
'G01 X6.322 Y6.818 Z0.000       ',
'G01 X6.817 Y6.335 Z0.000       ',
'G01 X7.275 Y5.815 Z0.000       ',
'G01 X7.692 Y5.262 Z0.000       ',
'G01 X8.068 Y4.679 Z-0.018      ',
'G01 X8.399 Y4.069 Z-0.142      ',
'G01 X8.685 Y3.436 Z-0.391      ',
'G01 X8.922 Y2.782 Z-0.786      ',
'G01 X9.109 Y2.112 Z-1.305      ',
'G01 X9.247 Y1.429 Z-1.799      ',
'G01 X9.333 Y0.737 Z-1.978      ',
'G01 X9.367 Y0.040 Z-2.125      ',
'G01 X9.352 Y-0.604 Z-2.003     ',
'G01 X9.292 Y-1.246 Z-1.748     ',
'G01 X9.189 Y-1.884 Z-1.375     ',
'G01 X9.041 Y-2.513 Z-0.968     ',
'G01 X8.850 Y-3.130 Z-0.526     ',
'G01 X8.617 Y-3.734 Z-0.230     ',
'G01 X8.343 Y-4.321 Z-0.061     ',
'G01 X8.029 Y-4.888 Z-0.008     ',
'G01 X7.675 Y-5.432 Z0.000      ',
'G01 X7.285 Y-5.951 Z0.000      ',
'G01 X6.860 Y-6.442 Z0.000      ',
'G01 X6.402 Y-6.903 Z0.000      ',
'G01 X5.912 Y-7.331 Z-0.035     ',
'G01 X5.394 Y-7.725 Z-0.165     ',
'G01 X4.849 Y-8.083 Z-0.413     ',
'G01 X4.280 Y-8.402 Z-0.718     ',
'G01 X3.690 Y-8.682 Z-1.135     ',
'G01 X3.082 Y-8.920 Z-1.512     ',
'G01 X2.459 Y-9.116 Z-2.052     ',
'G01 X1.823 Y-9.269 Z-2.696     ',
'G01 X1.177 Y-9.378 Z-3.207     ',
'G01 X0.525 Y-9.441 Z-3.207     ',
'G01 X0.525 Y-9.441 Z-4.092     ',
'G01 X-0.131 Y-9.460 Z-4.092    ',
'G01 X-0.131 Y-9.460 Z-4.869    ',
'G01 X-0.786 Y-9.433 Z-4.869    ',
'G01 X-0.786 Y-9.433 Z-5.782    ',
'G01 X-1.439 Y-9.361 Z-5.770    ',
'G01 X-2.086 Y-9.245 Z-5.772    ',
'G01 X-2.724 Y-9.083 Z-5.444    ',
'G01 X-3.349 Y-8.878 Z-5.214    ',
'G01 X-3.959 Y-8.630 Z-5.084    ',
'G01 X-4.552 Y-8.341 Z-5.041    ',
'G01 X-5.123 Y-8.010 Z-4.707    ',
'G01 X-5.670 Y-7.641 Z-4.808    ',
'G01 X-6.191 Y-7.235 Z-4.612    ',
'G01 X-6.684 Y-6.794 Z-4.479    ',
'G01 X-7.145 Y-6.319 Z-4.416    ',
'G01 X-7.572 Y-5.813 Z-4.233    ',
'G01 X-7.964 Y-5.278 Z-4.247    ',
'G01 X-8.318 Y-4.717 Z-4.176    ',
'G01 X-8.633 Y-4.133 Z-4.115    ',
'G01 X-8.907 Y-3.528 Z-3.995    ',
'G01 X-9.139 Y-2.905 Z-3.945    ',
'G01 X-9.328 Y-2.267 Z-3.967    ',
'G01 X-9.472 Y-1.617 Z-4.061    ',
'G01 X-9.571 Y-0.958 Z-4.000    ',
'G01 X-9.624 Y-0.293 Z-3.994    ',
'G01 X-9.631 Y0.374 Z-3.994     ',
'G01 X-9.592 Y1.041 Z-4.019     ',
'G01 X-9.508 Y1.704 Z-4.073     ',
'G01 X-9.377 Y2.360 Z-3.988     ',
'G01 X-9.202 Y3.006 Z-4.187     ',
'G01 X-8.982 Y3.639 Z-4.241     ',
'G01 X-8.719 Y4.255 Z-4.161     ',
'G01 X-8.414 Y4.853 Z-4.373     ',
'G01 X-8.068 Y5.428 Z-4.307     ',
'G01 X-7.682 Y5.979 Z-4.660     ',
'G01 X-7.260 Y6.502 Z-4.664     ',
'G01 X-6.802 Y6.995 Z-4.722     ',
'G01 X-6.311 Y7.455 Z-4.845     ',
'G01 X-5.788 Y7.881 Z-4.902     ',
'G01 X-5.237 Y8.270 Z-5.183     ',
'G01 X-4.661 Y8.621 Z-5.452     ',
'G01 X-4.060 Y8.931 Z-5.509     ',
'G01 X-3.440 Y9.199 Z-5.722     ',
'G01 X-2.802 Y9.424 Z-5.948     ',
'G01 X-2.149 Y9.604 Z-6.304     ',
'G01 X-1.486 Y9.739 Z-6.749     ',
'G01 X-0.814 Y9.828 Z-6.331     ',
'G01 X-0.814 Y9.828 Z-5.332     ',
'G01 X-0.136 Y9.870 Z-5.332     ',
'G01 X-0.136 Y9.870 Z-4.498     ',
'G01 X0.543 Y9.866 Z-4.498      ',
'G01 X1.220 Y9.815 Z-3.823      ',
'G01 X1.893 Y9.717 Z-3.265      ',
'G01 X1.893 Y9.717 Z-2.567      ',
'G01 X2.558 Y9.573 Z-2.567      ',
'G01 X3.212 Y9.383 Z-1.978      ',
'G01 X3.852 Y9.148 Z-1.481      ',
'G01 X4.474 Y8.869 Z-1.056      ',
'G01 X5.077 Y8.548 Z-0.544      ',
'G01 X5.656 Y8.186 Z-0.348      ',
'G01 X6.209 Y7.784 Z-0.122      ',
'G01 X6.733 Y7.345 Z-0.023      ',
'G01 X7.227 Y6.871 Z0.000       ',
'G01 X7.686 Y6.363 Z0.000       ',
'G01 X8.110 Y5.824 Z0.000       ',
'G01 X8.496 Y5.257 Z0.000       ',
'G01 X8.842 Y4.664 Z-0.008      ',
'G01 X9.147 Y4.048 Z-0.095      ',
'G01 X9.409 Y3.412 Z-0.286      ',
'G01 X9.626 Y2.759 Z-0.571      ',
'G01 X9.798 Y2.093 Z-0.937      ',
'G01 X9.924 Y1.415 Z-1.229      ',
'G01 X10.002 Y0.730 Z-1.531     ',
'G01 X10.033 Y0.040 Z-1.699     ',
'G01 X10.019 Y-0.607 Z-1.560    ',
'G01 X9.963 Y-1.253 Z-1.274     ',
'G01 X9.865 Y-1.895 Z-1.000     ',
'G01 X9.726 Y-2.529 Z-0.540     ',
'G01 X9.546 Y-3.153 Z-0.375     ',
'G01 X9.326 Y-3.765 Z-0.157     ',
'G01 X9.066 Y-4.361 Z-0.031     ',
'G01 X8.768 Y-4.940 Z-0.004     ',
'G01 X8.433 Y-5.499 Z0.000      ',
'G01 X8.063 Y-6.035 Z0.000      ',
'G01 X7.658 Y-6.546 Z0.000      ',
'G01 X7.220 Y-7.031 Z-0.001     ',
'G01 X6.752 Y-7.486 Z-0.041     ',
'G01 X6.255 Y-7.911 Z-0.164     ',
'G01 X5.731 Y-8.303 Z-0.389     ',
'G01 X5.183 Y-8.660 Z-0.640     ',
'G01 X4.612 Y-8.981 Z-1.106     ',
'G01 X4.021 Y-9.265 Z-1.518     ',
'G01 X3.412 Y-9.510 Z-2.005     ',
'G01 X2.789 Y-9.715 Z-2.585     ',
'G01 X2.153 Y-9.880 Z-3.111     ',
'G01 X1.508 Y-10.003 Z-3.615    ',
'G01 X0.855 Y-10.084 Z-3.615    ',
'G01 X0.855 Y-10.084 Z-4.533    ',
'G01 X0.198 Y-10.123 Z-4.533    ',
'G01 X0.198 Y-10.123 Z-5.320    ',
'G01 X-0.461 Y-10.119 Z-5.320   ',
'G01 X-0.461 Y-10.119 Z-6.333   ',
'G01 X-1.118 Y-10.073 Z-6.333   ',
'G01 X-1.118 Y-10.073 Z-7.000   ',
'G01 X-1.771 Y-9.984 Z-7.000    ',
'G01 X-2.418 Y-9.853 Z-7.000    ',
'G01 X-3.056 Y-9.680 Z-6.682    ',
'G01 X-3.681 Y-9.466 Z-6.420    ',
'G01 X-4.291 Y-9.212 Z-6.189    ',
'G01 X-4.884 Y-8.919 Z-5.771    ',
'G01 X-5.458 Y-8.587 Z-5.829    ',
'G01 X-6.009 Y-8.219 Z-5.499    ',
'G01 X-6.535 Y-7.816 Z-5.437    ',
'G01 X-7.035 Y-7.379 Z-5.284    ',
'G01 X-7.505 Y-6.911 Z-5.208    ',
'G01 X-7.945 Y-6.413 Z-5.197    ',
'G01 X-8.351 Y-5.887 Z-5.203    ',
'G01 X-8.723 Y-5.335 Z-4.846    ',
'G01 X-9.059 Y-4.760 Z-4.980    ',
'G01 X-9.357 Y-4.165 Z-4.780    ',
'G01 X-9.616 Y-3.550 Z-4.668    ',
'G01 X-9.834 Y-2.920 Z-4.607    ',
'G01 X-10.012 Y-2.277 Z-4.517   ',
'G01 X-10.148 Y-1.623 Z-4.403   ',
'G01 X-10.241 Y-0.961 Z-4.373   ',
'G01 X-10.291 Y-0.294 Z-4.358   ',
'G01 X-10.298 Y0.375 Z-4.358    ',
'G01 X-10.262 Y1.044 Z-4.378    ',
'G01 X-10.182 Y1.709 Z-4.436    ',
'G01 X-10.059 Y2.369 Z-4.531    ',
'G01 X-9.894 Y3.019 Z-4.705     ',
'G01 X-9.687 Y3.658 Z-4.937     ',
'G01 X-9.438 Y4.282 Z-5.087     ',
'G01 X-9.150 Y4.889 Z-5.041     ',
'G01 X-8.823 Y5.477 Z-5.148     ',
'G01 X-8.458 Y6.043 Z-5.284     ',
'G01 X-8.057 Y6.584 Z-5.282     ',
'G01 X-7.621 Y7.099 Z-5.541     ',
'G01 X-7.153 Y7.585 Z-5.650     ',
'G01 X-6.654 Y8.039 Z-5.835     ',
'G01 X-6.126 Y8.461 Z-6.116     ',
'G01 X-5.572 Y8.848 Z-6.324     ',
'G01 X-4.993 Y9.198 Z-6.412     ',
'G01 X-4.393 Y9.511 Z-6.896     ',
'G01 X-3.773 Y9.784 Z-7.000     ',
'G01 X-3.137 Y10.016 Z-7.000    ',
'G01 X-2.486 Y10.207 Z-7.000    ',
'G01 X-1.824 Y10.356 Z-7.000    ',
'G01 X-1.153 Y10.461 Z-7.000    ',
'G01 X-0.476 Y10.523 Z-7.000    ',
'G01 X-0.476 Y10.523 Z-5.854    ',
'G01 X0.203 Y10.541 Z-5.854     ',
'G01 X0.203 Y10.541 Z-4.997     ',
'G01 X0.883 Y10.515 Z-4.997     ',
'G01 X1.560 Y10.444 Z-4.320     ',
'G01 X1.560 Y10.444 Z-3.480     ',
'G01 X2.232 Y10.330 Z-3.480     ',
'G01 X2.895 Y10.173 Z-3.044     ',
'G01 X3.548 Y9.973 Z-2.435      ',
'G01 X4.186 Y9.731 Z-1.929      ',
'G01 X4.808 Y9.448 Z-1.363      ',
'G01 X5.410 Y9.125 Z-1.000      ',
'G01 X5.991 Y8.764 Z-0.538      ',
'G01 X6.547 Y8.365 Z-0.262      ',
'G01 X7.077 Y7.931 Z-0.156      ',
'G01 X7.578 Y7.464 Z-0.016      ',
'G01 X8.048 Y6.964 Z0.000       ',
'G01 X8.485 Y6.435 Z0.000       ',
'G01 X8.887 Y5.879 Z0.000       ',
'G01 X9.252 Y5.297 Z0.000       ',
'G01 X9.579 Y4.692 Z0.000       ',
'G01 X9.866 Y4.067 Z-0.045      ',
'G01 X10.113 Y3.424 Z-0.170     ',
'G01 X10.317 Y2.766 Z-0.357     ',
'G01 X10.479 Y2.096 Z-0.552     ',
'G01 X10.597 Y1.417 Z-0.678     ',
'G01 X10.671 Y0.730 Z-0.914     ',
'G01 X10.700 Y0.040 Z-1.083     ',
'G01 X10.687 Y-0.610 Z-0.939    ',
'G01 X10.634 Y-1.259 Z-0.708    ',
'G01 X10.541 Y-1.904 Z-0.587    ',
'G01 X10.409 Y-2.543 Z-0.322    ',
'G01 X10.239 Y-3.172 Z-0.224    ',
'G01 X10.030 Y-3.791 Z-0.082    ',
'G01 X9.783 Y-4.396 Z-0.009     ',
'G01 X9.501 Y-4.985 Z0.000      ',
'G01 X9.182 Y-5.556 Z0.000      ',
'G01 X8.829 Y-6.107 Z0.000      ',
'G01 X8.443 Y-6.636 Z0.000      ',
'G01 X8.025 Y-7.141 Z0.000      ',
'G01 X7.577 Y-7.619 Z-0.034     ',
'G01 X7.100 Y-8.070 Z-0.132     ',
'G01 X6.597 Y-8.491 Z-0.314     ',
'G01 X6.068 Y-8.880 Z-0.638     ',
'G01 X5.516 Y-9.237 Z-1.073     ',
'G01 X4.943 Y-9.560 Z-1.427     ',
'G01 X4.352 Y-9.847 Z-1.849     ',
'G01 X3.743 Y-10.098 Z-2.488    ',
'G01 X3.120 Y-10.312 Z-3.084    ',
'G01 X2.484 Y-10.487 Z-3.501    ',
'G01 X1.839 Y-10.623 Z-3.501    ',
'G01 X1.839 Y-10.623 Z-4.327    ',
'G01 X1.186 Y-10.720 Z-4.984    ',
'G01 X0.529 Y-10.777 Z-4.984    ',
'G01 X0.529 Y-10.777 Z-6.258    ',
'G01 X-0.132 Y-10.793 Z-6.258   ',
'G01 X-0.132 Y-10.793 Z-7.000   ',
'G01 X-0.793 Y-10.769 Z-7.000   ',
'G01 X-1.451 Y-10.705 Z-7.000   ',
'G01 X-2.105 Y-10.601 Z-7.000   ',
'G01 X-2.751 Y-10.457 Z-7.000   ',
'G01 X-3.388 Y-10.274 Z-7.000   ',
'G01 X-4.013 Y-10.053 Z-7.000   ',
'G01 X-4.623 Y-9.793 Z-7.000    ',
'G01 X-5.217 Y-9.496 Z-7.000    ',
'G01 X-5.792 Y-9.164 Z-6.762    ',
'G01 X-6.346 Y-8.797 Z-6.981    ',
'G01 X-6.877 Y-8.397 Z-6.626    ',
'G01 X-7.383 Y-7.964 Z-6.391    ',
'G01 X-7.862 Y-7.502 Z-6.544    ',
'G01 X-8.312 Y-7.011 Z-6.511    ',
'G01 X-8.732 Y-6.493 Z-5.927    ',
'G01 X-9.119 Y-5.950 Z-5.983    ',
'G01 X-9.473 Y-5.384 Z-5.900    ',
'G01 X-9.792 Y-4.797 Z-5.729    ',
'G01 X-10.074 Y-4.192 Z-5.250   ',
'G01 X-10.320 Y-3.570 Z-4.875   ',
'G01 X-10.527 Y-2.933 Z-4.625   ',
'G01 X-10.695 Y-2.286 Z-4.466   ',
'G01 X-10.823 Y-1.628 Z-4.396   ',
'G01 X-10.911 Y-0.964 Z-4.356   ',
'G01 X-10.958 Y-0.295 Z-4.354   ',
'G01 X-10.965 Y0.376 Z-4.354    ',
'G01 X-10.930 Y1.046 Z-4.358    ',
'G01 X-10.855 Y1.714 Z-4.407    ',
'G01 X-10.739 Y2.376 Z-4.528    ',
'G01 X-10.583 Y3.030 Z-4.651    ',
'G01 X-10.387 Y3.674 Z-4.910    ',
'G01 X-10.152 Y4.305 Z-5.270    ',
'G01 X-9.879 Y4.921 Z-5.751     ',
'G01 X-9.569 Y5.519 Z-6.210     ',
'G01 X-9.222 Y6.098 Z-6.392     ',
'G01 X-8.841 Y6.655 Z-6.630     ',
'G01 X-8.426 Y7.188 Z-6.630     ',
'G01 X-7.979 Y7.695 Z-6.668     ',
'G01 X-7.502 Y8.174 Z-7.000     ',
'G01 X-6.996 Y8.623 Z-7.000     ',
'G01 X-6.464 Y9.041 Z-7.000     ',
'G01 X-5.907 Y9.425 Z-7.000     ',
'G01 X-5.326 Y9.776 Z-7.000     ',
'G01 X-4.726 Y10.090 Z-7.000    ',
'G01 X-4.107 Y10.368 Z-7.000    ',
'G01 X-3.471 Y10.607 Z-7.000    ',
'G01 X-2.822 Y10.807 Z-7.000    ',
'G01 X-2.162 Y10.968 Z-7.000    ',
'G01 X-1.493 Y11.088 Z-7.000    ',
'G01 X-0.817 Y11.167 Z-7.000    ',
'G01 X-0.137 Y11.204 Z-7.000    ',
'G01 X-0.137 Y11.204 Z-6.977    ',
'G01 X0.544 Y11.200 Z-6.977     ',
'G01 X0.544 Y11.200 Z-5.951     ',
'G01 X1.224 Y11.155 Z-5.951     ',
'G01 X1.224 Y11.155 Z-5.181     ',
'G01 X1.901 Y11.068 Z-5.181     ',
'G01 X1.901 Y11.068 Z-4.228     ',
'G01 X2.571 Y10.940 Z-4.228     ',
'G01 X2.571 Y10.940 Z-3.468     ',
'G01 X3.233 Y10.771 Z-3.468     ',
'G01 X3.883 Y10.562 Z-2.834     ',
'G01 X4.520 Y10.314 Z-2.308     ',
'G01 X5.141 Y10.027 Z-1.869     ',
'G01 X5.744 Y9.703 Z-1.291      ',
'G01 X6.326 Y9.342 Z-1.030      ',
'G01 X6.885 Y8.946 Z-0.611      ',
'G01 X7.419 Y8.517 Z-0.332      ',
'G01 X7.927 Y8.055 Z-0.152      ',
'G01 X8.406 Y7.563 Z-0.044      ',
'G01 X8.854 Y7.043 Z-0.004      ',
'G01 X9.270 Y6.496 Z0.000       ',
'G01 X9.651 Y5.924 Z0.000       ',
'G01 X9.998 Y5.330 Z0.000       ',
'G01 X10.308 Y4.715 Z0.000      ',
'G01 X10.580 Y4.083 Z-0.010     ',
'G01 X10.813 Y3.434 Z-0.046     ',
'G01 X11.006 Y2.772 Z-0.172     ',
'G01 X11.158 Y2.099 Z-0.257     ',
'G01 X11.270 Y1.418 Z-0.313     ',
'G01 X11.339 Y0.731 Z-0.435     ',
'G01 X11.367 Y0.040 Z-0.520     ',
'G01 X11.354 Y-0.613 Z-0.448    ',
'G01 X11.304 Y-1.265 Z-0.329    ',
'G01 X11.216 Y-1.913 Z-0.274    ',
'G01 X11.091 Y-2.555 Z-0.136    ',
'G01 X10.929 Y-3.190 Z-0.059    ',
'G01 X10.730 Y-3.814 Z-0.024    ',
'G01 X10.496 Y-4.426 Z0.000     ',
'G01 X10.227 Y-5.024 Z0.000     ',
'G01 X9.923 Y-5.606 Z0.000      ',
'G01 X9.587 Y-6.170 Z0.000      ',
'G01 X9.218 Y-6.714 Z0.000      ',
'G01 X8.818 Y-7.236 Z-0.010     ',
'G01 X8.389 Y-7.734 Z-0.073     ',
'G01 X7.931 Y-8.207 Z-0.200     ',
'G01 X7.447 Y-8.653 Z-0.403     ',
'G01 X6.938 Y-9.070 Z-0.715     ',
'G01 X6.405 Y-9.458 Z-1.127     ',
'G01 X5.850 Y-9.814 Z-1.424     ',
'G01 X5.275 Y-10.139 Z-1.955    ',
'G01 X4.683 Y-10.429 Z-2.386    ',
'G01 X4.074 Y-10.685 Z-2.902    ',
'G01 X3.451 Y-10.906 Z-3.524    ',
'G01 X2.816 Y-11.091 Z-4.119    ',
'G01 X2.171 Y-11.239 Z-4.119    ',
'G01 X2.171 Y-11.239 Z-5.008    ',
'G01 X1.519 Y-11.349 Z-5.008    ',
'G01 X1.519 Y-11.349 Z-5.687    ',
'G01 X0.861 Y-11.422 Z-5.687    ',
'G01 X0.861 Y-11.422 Z-7.000    ',
'G01 X0.199 Y-11.457 Z-7.000    ',
'G01 X-0.464 Y-11.453 Z-7.000   ',
'G01 X-1.126 Y-11.412 Z-7.000   ',
'G01 X-1.785 Y-11.332 Z-7.000   ',
'G01 X-2.438 Y-11.214 Z-7.000   ',
'G01 X-3.084 Y-11.059 Z-7.000   ',
'G01 X-3.720 Y-10.867 Z-7.000   ',
'G01 X-4.345 Y-10.638 Z-7.000   ',
'G01 X-4.955 Y-10.374 Z-7.000   ',
'G01 X-5.550 Y-10.074 Z-7.000   ',
'G01 X-6.127 Y-9.741 Z-7.000    ',
'G01 X-6.684 Y-9.375 Z-7.000    ',
'G01 X-7.219 Y-8.977 Z-7.000    ',
'G01 X-7.730 Y-8.549 Z-7.000    ',
'G01 X-8.217 Y-8.092 Z-7.000    ',
'G01 X-8.676 Y-7.607 Z-7.000    ',
'G01 X-9.107 Y-7.096 Z-7.000    ',
'G01 X-9.508 Y-6.561 Z-7.000    ',
'G01 X-9.508 Y-6.561 Z-6.750    ',
'G01 X-9.878 Y-6.004 Z-6.750    ',
'G01 X-10.215 Y-5.425 Z-6.228   ',
'G01 X-10.518 Y-4.829 Z-5.635   ',
'G01 X-10.787 Y-4.215 Z-5.191   ',
'G01 X-11.020 Y-3.586 Z-4.863   ',
'G01 X-11.216 Y-2.945 Z-4.623   ',
'G01 X-11.376 Y-2.293 Z-4.510   ',
'G01 X-11.497 Y-1.633 Z-4.396   ',
'G01 X-11.581 Y-0.966 Z-4.356   ',
'G01 X-11.625 Y-0.296 Z-4.354   ',
'G01 X-11.632 Y0.377 Z-4.354    ',
'G01 X-11.599 Y1.049 Z-4.358    ',
'G01 X-11.528 Y1.718 Z-4.407    ',
'G01 X-11.418 Y2.383 Z-4.526    ',
'G01 X-11.270 Y3.040 Z-4.650    ',
'G01 X-11.084 Y3.688 Z-4.898    ',
'G01 X-10.861 Y4.325 Z-5.236    ',
'G01 X-10.602 Y4.948 Z-5.687    ',
'G01 X-10.307 Y5.555 Z-6.286    ',
'G01 X-9.977 Y6.145 Z-6.851     ',
'G01 X-9.614 Y6.715 Z-6.851     ',
'G01 X-9.614 Y6.715 Z-7.000     ',
'G01 X-9.218 Y7.264 Z-7.000     ',
'G01 X-8.791 Y7.789 Z-7.000     ',
'G01 X-8.334 Y8.288 Z-7.000     ',
'G01 X-7.849 Y8.761 Z-7.000     ',
'G01 X-7.338 Y9.206 Z-7.000     ',
'G01 X-6.801 Y9.620 Z-7.000     ',
'G01 X-6.241 Y10.003 Z-7.000    ',
'G01 X-5.659 Y10.353 Z-7.000    ',
'G01 X-5.059 Y10.670 Z-7.000    ',
'G01 X-4.440 Y10.951 Z-7.000    ',
'G01 X-3.806 Y11.196 Z-7.000    ',
'G01 X-3.159 Y11.405 Z-7.000    ',
'G01 X-2.500 Y11.576 Z-7.000    ',
'G01 X-1.832 Y11.709 Z-7.000    ',
'G01 X-1.157 Y11.803 Z-7.000    ',
'G01 X-0.478 Y11.858 Z-7.000    ',
'G01 X0.204 Y11.874 Z-7.000     ',
'G01 X0.886 Y11.851 Z-7.000     ',
'G01 X0.886 Y11.851 Z-6.919     ',
'G01 X1.566 Y11.788 Z-6.919     ',
'G01 X1.566 Y11.788 Z-5.577     ',
'G01 X2.241 Y11.686 Z-5.577     ',
'G01 X2.910 Y11.546 Z-4.983     ',
'G01 X2.910 Y11.546 Z-4.150     ',
'G01 X3.570 Y11.367 Z-4.150     ',
'G01 X4.218 Y11.150 Z-3.486     ',
'G01 X4.854 Y10.896 Z-2.934     ',
'G01 X5.474 Y10.606 Z-2.533     ',
'G01 X6.077 Y10.280 Z-1.901     ',
'G01 X6.660 Y9.920 Z-1.378      ',
'G01 X7.222 Y9.526 Z-1.148      ',
'G01 X7.761 Y9.101 Z-0.760      ',
'G01 X8.274 Y8.645 Z-0.449      ',
'G01 X8.761 Y8.160 Z-0.232      ',
'G01 X9.219 Y7.648 Z-0.047      ',
'G01 X9.647 Y7.110 Z-0.006      ',
'G01 X10.043 Y6.548 Z0.000      ',
'G01 X10.407 Y5.963 Z0.000      ',
'G01 X10.736 Y5.358 Z0.000      ',
'G01 X11.030 Y4.735 Z0.000      ',
'G01 X11.288 Y4.096 Z0.000      ',
'G01 X11.509 Y3.443 Z-0.004     ',
'G01 X11.692 Y2.777 Z-0.042     ',
'G01 X11.836 Y2.102 Z-0.076     ',
'G01 X11.942 Y1.419 Z-0.094     ',
'G01 X12.007 Y0.731 Z-0.152     ',
'G01 X12.033 Y0.040 Z-0.193     ',
'G01 X12.021 Y-0.610 Z-0.158    ',
'G01 X11.974 Y-1.258 Z-0.100    ',
'G01 X11.892 Y-1.904 Z-0.085    ',
'G01 X11.775 Y-2.544 Z-0.025    ',
'G01 X11.624 Y-3.178 Z-0.015    ',
'G01 X11.438 Y-3.802 Z0.000     ',
'G01 X11.218 Y-4.416 Z0.000     ',
'G01 X10.966 Y-5.018 Z0.000     ',
'G01 X10.681 Y-5.605 Z0.000     ',
'G01 X10.365 Y-6.176 Z0.000     ',
'G01 X10.018 Y-6.729 Z0.000     ',
'G01 X9.641 Y-7.263 Z-0.014     ',
'G01 X9.236 Y-7.777 Z-0.077     ',
'G01 X8.804 Y-8.267 Z-0.200     ',
'G01 X8.345 Y-8.734 Z-0.400     ',
'G01 X7.861 Y-9.176 Z-0.694     ',
'G01 X7.355 Y-9.590 Z-1.070     ',
'G01 X6.826 Y-9.977 Z-1.495     ',
'G01 X6.276 Y-10.335 Z-2.013    ',
'G01 X5.708 Y-10.663 Z-2.337    ',
'G01 X5.123 Y-10.960 Z-2.337    ',
'G01 X5.123 Y-10.960 Z-3.043    ',
'G01 X4.522 Y-11.225 Z-3.587    ',
'G01 X3.907 Y-11.457 Z-3.587    ',
'G01 X3.907 Y-11.457 Z-4.248    ',
'G01 X3.281 Y-11.655 Z-4.248    ',
'G01 X3.281 Y-11.655 Z-4.908    ',
'G01 X2.644 Y-11.819 Z-5.442    ',
'G01 X1.999 Y-11.949 Z-5.442    ',
'G01 X1.999 Y-11.949 Z-6.663    ',
'G01 X1.348 Y-12.043 Z-6.663    ',
'G01 X1.348 Y-12.043 Z-7.000    ',
'G01 X0.692 Y-12.103 Z-7.000    ',
'G01 X0.033 Y-12.126 Z-7.000    ',
'G01 X-0.626 Y-12.114 Z-7.000   ',
'G01 X-1.283 Y-12.066 Z-7.000   ',
'G01 X-1.938 Y-11.983 Z-7.000   ',
'G01 X-2.587 Y-11.864 Z-7.000   ',
'G01 X-3.229 Y-11.710 Z-7.000   ',
'G01 X-3.863 Y-11.522 Z-7.000   ',
'G01 X-4.485 Y-11.299 Z-7.000   ',
'G01 X-5.095 Y-11.043 Z-7.000   ',
'G01 X-5.690 Y-10.755 Z-7.000   ',
'G01 X-6.269 Y-10.434 Z-7.000   ',
'G01 X-6.830 Y-10.082 Z-7.000   ',
'G01 X-7.371 Y-9.700 Z-7.000    ',
'G01 X-7.892 Y-9.289 Z-7.000    ',
'G01 X-8.389 Y-8.851 Z-7.000    ',
'G01 X-8.862 Y-8.386 Z-7.000    ',
'G01 X-9.310 Y-7.896 Z-7.000    ',
'G01 X-9.730 Y-7.382 Z-7.000    ',
'G01 X-10.123 Y-6.845 Z-7.000   ',
'G01 X-10.123 Y-6.845 Z-6.961   ',
'G01 X-10.485 Y-6.288 Z-6.961   ',
'G01 X-10.818 Y-5.712 Z-6.414   ',
'G01 X-11.118 Y-5.119 Z-5.795   ',
'G01 X-11.387 Y-4.510 Z-5.323   ',
'G01 X-11.622 Y-3.887 Z-5.071   ',
'G01 X-11.823 Y-3.251 Z-4.775   ',
'G01 X-11.989 Y-2.606 Z-4.564   ',
'G01 X-12.121 Y-1.952 Z-4.434   ',
'G01 X-12.216 Y-1.292 Z-4.368   ',
'G01 X-12.276 Y-0.627 Z-4.356   ',
'G01 X-12.300 Y0.040 Z-4.356    ',
'G01 X-12.288 Y0.708 Z-4.356    ',
'G01 X-12.239 Y1.375 Z-4.373    ',
'G01 X-12.155 Y2.039 Z-4.446    ',
'G01 X-12.034 Y2.697 Z-4.586    ',
'G01 X-11.878 Y3.348 Z-4.808    ',
'G01 X-11.687 Y3.990 Z-5.114    ',
'G01 X-11.461 Y4.620 Z-5.523    ',
'G01 X-11.202 Y5.238 Z-5.859    ',
'G01 X-10.909 Y5.842 Z-6.505    ',
'G01 X-10.584 Y6.429 Z-6.505    ',
'G01 X-10.584 Y6.429 Z-7.000    ',
'G01 X-10.227 Y6.997 Z-7.000    ',
'G01 X-9.840 Y7.546 Z-7.000     ',
'G01 X-9.424 Y8.073 Z-7.000     ',
'G01 X-8.979 Y8.577 Z-7.000     ',
'G01 X-8.508 Y9.057 Z-7.000     ',
'G01 X-8.011 Y9.511 Z-7.000     ',
'G01 X-7.490 Y9.937 Z-7.000     ',
'G01 X-6.946 Y10.334 Z-7.000    ',
'G01 X-6.381 Y10.702 Z-7.000    ',
'G01 X-5.798 Y11.039 Z-7.000    ',
'G01 X-5.196 Y11.343 Z-7.000    ',
'G01 X-4.579 Y11.615 Z-7.000    ',
'G01 X-3.947 Y11.853 Z-7.000    ',
'G01 X-3.303 Y12.057 Z-7.000    ',
'G01 X-2.649 Y12.226 Z-7.000    ',
'G01 X-1.986 Y12.359 Z-7.000    ',
'G01 X-1.317 Y12.456 Z-7.000    ',
'G01 X-0.643 Y12.516 Z-7.000    ',
'G01 X0.033 Y12.540 Z-7.000     ',
'G01 X0.710 Y12.528 Z-7.000     ',
'G01 X1.386 Y12.479 Z-7.000     ',
'G01 X2.058 Y12.393 Z-7.000     ',
'G01 X2.058 Y12.393 Z-6.634     ',
'G01 X2.725 Y12.271 Z-6.634     ',
'G01 X2.725 Y12.271 Z-5.491     ',
'G01 X3.385 Y12.113 Z-5.491     ',
'G01 X3.385 Y12.113 Z-4.626     ',
'G01 X4.036 Y11.919 Z-4.626     ',
'G01 X4.036 Y11.919 Z-3.944     ',
'G01 X4.675 Y11.690 Z-3.944     ',
'G01 X5.301 Y11.427 Z-3.382     ',
'G01 X5.913 Y11.130 Z-2.972     ',
'G01 X6.507 Y10.800 Z-2.318     ',
'G01 X7.084 Y10.439 Z-2.014     ',
'G01 X7.640 Y10.047 Z-1.552     ',
'G01 X8.174 Y9.624 Z-1.139      ',
'G01 X8.685 Y9.174 Z-0.760      ',
'G01 X9.171 Y8.696 Z-0.459      ',
'G01 X9.630 Y8.192 Z-0.256      ',
'G01 X10.062 Y7.664 Z-0.073     ',
'G01 X10.465 Y7.113 Z-0.021     ',
'G01 X10.838 Y6.541 Z0.000      ',
'G01 X11.179 Y5.949 Z0.000      ',
'G01 X11.488 Y5.340 Z0.000      ',
'G01 X11.763 Y4.714 Z0.000      ',
'G01 X12.004 Y4.074 Z0.000      ',
'G01 X12.211 Y3.421 Z0.000      ',
'G01 X12.381 Y2.758 Z0.000      ',
'G01 X12.516 Y2.087 Z-0.004     ',
'G01 X12.614 Y1.409 Z-0.006     ',
'G01 X12.676 Y0.726 Z-0.018     ',
'G01 X12.700 Y0.040 Z-0.032     ',
'G01 X12.689 Y-0.612 Z-0.020    ',
'G01 X12.644 Y-1.263 Z-0.007    ',
'G01 X12.565 Y-1.911 Z-0.005    ',
'G01 X12.454 Y-2.555 Z0.000     ',
'G01 X12.309 Y-3.192 Z0.000     ',
'G01 X12.131 Y-3.822 Z0.000     ',
'G01 X11.922 Y-4.441 Z0.000     ',
'G01 X11.680 Y-5.049 Z0.000     ',
'G01 X11.407 Y-5.645 Z0.000     ',
'G01 X11.105 Y-6.225 Z0.000     ',
'G01 X10.772 Y-6.790 Z-0.005    ',
'G01 X10.410 Y-7.337 Z-0.038    ',
'G01 X10.021 Y-7.865 Z-0.168    ',
'G01 X9.605 Y-8.372 Z-0.320     ',
'G01 X9.163 Y-8.857 Z-0.546     ',
'G01 X8.697 Y-9.320 Z-0.876     ',
'G01 X8.207 Y-9.757 Z-1.264     ',
'G01 X7.695 Y-10.170 Z-1.689    ',
'G01 X7.162 Y-10.555 Z-2.171    ',
'G01 X6.610 Y-10.913 Z-2.454    ',
'G01 X6.040 Y-11.241 Z-3.112    ',
'G01 X5.454 Y-11.541 Z-3.584    ',
'G01 X4.853 Y-11.809 Z-4.071    ',
'G01 X4.238 Y-12.047 Z-4.071    ',
'G01 X4.238 Y-12.047 Z-4.755    ',
'G01 X3.612 Y-12.253 Z-4.755    ',
'G01 X3.612 Y-12.253 Z-5.617    ',
'G01 X2.975 Y-12.426 Z-5.617    ',
'G01 X2.975 Y-12.426 Z-6.782    ',
'G01 X2.331 Y-12.566 Z-6.782    ',
'G01 X2.331 Y-12.566 Z-7.000    ',
'G01 X1.679 Y-12.673 Z-7.000    ',
'G01 X1.023 Y-12.746 Z-7.000    ',
'G01 X0.364 Y-12.786 Z-7.000    ',
'G01 X-0.297 Y-12.791 Z-7.000   ',
'G01 X-0.958 Y-12.763 Z-7.000   ',
'G01 X-1.616 Y-12.700 Z-7.000   ',
'G01 X-2.271 Y-12.604 Z-7.000   ',
'G01 X-2.920 Y-12.474 Z-7.000   ',
'G01 X-3.562 Y-12.310 Z-7.000   ',
'G01 X-4.195 Y-12.114 Z-7.000   ',
'G01 X-4.817 Y-11.885 Z-7.000   ',
'G01 X-5.427 Y-11.625 Z-7.000   ',
'G01 X-6.022 Y-11.333 Z-7.000   ',
'G01 X-6.603 Y-11.011 Z-7.000   ',
'G01 X-7.166 Y-10.659 Z-7.000   ',
'G01 X-7.710 Y-10.279 Z-7.000   ',
'G01 X-8.235 Y-9.871 Z-7.000    ',
'G01 X-8.738 Y-9.436 Z-7.000    ',
'G01 X-9.218 Y-8.976 Z-7.000    ',
'G01 X-9.674 Y-8.491 Z-7.000    ',
'G01 X-10.105 Y-7.983 Z-7.000   ',
'G01 X-10.509 Y-7.454 Z-7.000   ',
'G01 X-10.885 Y-6.904 Z-7.000   ',
'G01 X-11.233 Y-6.336 Z-7.000   ',
'G01 X-11.233 Y-6.336 Z-6.414   ',
'G01 X-11.551 Y-5.750 Z-6.414   ',
'G01 X-11.839 Y-5.148 Z-5.795   ',
'G01 X-12.095 Y-4.532 Z-5.475   ',
'G01 X-12.320 Y-3.903 Z-5.095   ',
'G01 X-12.512 Y-3.263 Z-4.798   ',
'G01 X-12.670 Y-2.614 Z-4.607   ',
'G01 X-12.796 Y-1.958 Z-4.500   ',
'G01 X-12.887 Y-1.295 Z-4.419   ',
'G01 X-12.944 Y-0.628 Z-4.377   ',
'G01 X-12.967 Y0.040 Z-4.396    ',
'G01 X-12.955 Y0.710 Z-4.379    ',
'G01 X-12.909 Y1.378 Z-4.426    ',
'G01 X-12.828 Y2.044 Z-4.512    ',
'G01 X-12.713 Y2.704 Z-4.627    ',
'G01 X-12.564 Y3.358 Z-4.852    ',
'G01 X-12.382 Y4.004 Z-5.138    ',
'G01 X-12.167 Y4.640 Z-5.531    ',
'G01 X-11.919 Y5.264 Z-6.058    ',
'G01 X-11.639 Y5.875 Z-6.505    ',
'G01 X-11.328 Y6.470 Z-6.505    ',
'G01 X-11.328 Y6.470 Z-7.000    ',
'G01 X-10.986 Y7.050 Z-7.000    ',
'G01 X-10.615 Y7.611 Z-7.000    ',
'G01 X-10.216 Y8.152 Z-7.000    ',
'G01 X-9.789 Y8.673 Z-7.000     ',
'G01 X-9.335 Y9.171 Z-7.000     ',
'G01 X-8.857 Y9.645 Z-7.000     ',
'G01 X-8.354 Y10.094 Z-7.000    ',
'G01 X-7.828 Y10.517 Z-7.000    ',
'G01 X-7.282 Y10.912 Z-7.000    ',
'G01 X-6.715 Y11.279 Z-7.000    ',
'G01 X-6.130 Y11.617 Z-7.000    ',
'G01 X-5.529 Y11.923 Z-7.000    ',
'G01 X-4.911 Y12.199 Z-7.000    ',
'G01 X-4.281 Y12.443 Z-7.000    ',
'G01 X-3.638 Y12.654 Z-7.000    ',
'G01 X-2.985 Y12.831 Z-7.000    ',
'G01 X-2.324 Y12.975 Z-7.000    ',
'G01 X-1.655 Y13.085 Z-7.000    ',
'G01 X-0.982 Y13.160 Z-7.000    ',
'G01 X-0.306 Y13.200 Z-7.000    ',
'G01 X0.372 Y13.205 Z-7.000     ',
'G01 X1.050 Y13.176 Z-7.000     ',
'G01 X1.726 Y13.112 Z-7.000     ',
'G01 X2.397 Y13.013 Z-7.000     ',
'G01 X3.063 Y12.879 Z-7.000     ',
'G01 X3.063 Y12.879 Z-6.727     ',
'G01 X3.722 Y12.711 Z-6.727     ',
'G01 X3.722 Y12.711 Z-5.679     ',
'G01 X4.371 Y12.510 Z-5.679     ',
'G01 X4.371 Y12.510 Z-4.991     ',
'G01 X5.009 Y12.275 Z-4.991     ',
'G01 X5.635 Y12.008 Z-4.343     ',
'G01 X6.246 Y11.708 Z-3.819     ',
'G01 X6.246 Y11.708 Z-3.098     ',
'G01 X6.841 Y11.378 Z-3.098     ',
'G01 X7.419 Y11.017 Z-2.511     ',
'G01 X7.977 Y10.626 Z-2.252     ',
'G01 X8.515 Y10.208 Z-1.773     ',
'G01 X9.031 Y9.761 Z-1.344      ',
'G01 X9.523 Y9.289 Z-0.990      ',
'G01 X9.991 Y8.792 Z-0.523      ',
'G01 X10.433 Y8.271 Z-0.331     ',
'G01 X10.847 Y7.728 Z-0.202     ',
'G01 X11.233 Y7.164 Z-0.052     ',
'G01 X11.590 Y6.581 Z-0.006     ',
'G01 X11.916 Y5.980 Z0.000      ',
'G01 X12.211 Y5.362 Z0.000      ',
'G01 X12.474 Y4.730 Z0.000      ',
'G01 X12.704 Y4.085 Z0.000      ',
'G01 X12.901 Y3.429 Z0.000      ',
'G01 X13.063 Y2.763 Z0.000      ',
'G01 X13.192 Y2.090 Z0.000      ',
'G01 X13.285 Y1.410 Z0.000      ',
'G01 X13.344 Y0.727 Z0.000      ',
'G01 X13.367 Y0.040 Z0.000      ',
'G01 X13.356 Y-0.614 Z0.000     ',
'G01 X13.313 Y-1.267 Z0.000     ',
'G01 X13.238 Y-1.918 Z0.000     ',
'G01 X13.131 Y-2.565 Z0.000     ',
'G01 X12.992 Y-3.206 Z0.000     ',
'G01 X12.822 Y-3.839 Z0.000     ',
'G01 X12.622 Y-4.464 Z0.000     ',
'G01 X12.390 Y-5.078 Z0.000     ',
'G01 X12.129 Y-5.680 Z0.000     ',
'G01 X11.838 Y-6.269 Z0.000     ',
'G01 X11.519 Y-6.844 Z-0.037    ',
'G01 X11.172 Y-7.402 Z-0.079    ',
'G01 X10.797 Y-7.943 Z-0.228    ',
'G01 X10.397 Y-8.464 Z-0.400    ',
'G01 X9.971 Y-8.966 Z-0.790     ',
'G01 X9.520 Y-9.447 Z-1.114     ',
'G01 X9.047 Y-9.904 Z-1.487     ',
'G01 X8.551 Y-10.339 Z-1.920    ',
'G01 X8.035 Y-10.748 Z-2.412    ',
'G01 X7.499 Y-11.132 Z-2.682    ',
'G01 X6.944 Y-11.490 Z-3.287    ',
'G01 X6.373 Y-11.820 Z-3.661    ',
'G01 X5.785 Y-12.121 Z-3.661    ',
'G01 X5.785 Y-12.121 Z-4.521    ',
'G01 X5.184 Y-12.393 Z-5.169    ',
'G01 X4.569 Y-12.636 Z-5.169    ',
'G01 X4.569 Y-12.636 Z-6.009    ',
'G01 X3.943 Y-12.848 Z-6.009    ',
'G01 X3.943 Y-12.848 Z-6.942    ',
'G01 X3.307 Y-13.030 Z-6.942    ',
'G01 X3.307 Y-13.030 Z-7.000    ',
'G01 X2.663 Y-13.180 Z-7.000    ',
'G01 X2.012 Y-13.298 Z-7.000    ',
'G01 X1.356 Y-13.384 Z-7.000    ',
'G01 X0.695 Y-13.438 Z-7.000    ',
'G01 X0.033 Y-13.460 Z-7.000    ',
'G01 X-0.629 Y-13.448 Z-7.000   ',
'G01 X-1.291 Y-13.405 Z-7.000   ',
'G01 X-1.950 Y-13.329 Z-7.000   ',
'G01 X-2.604 Y-13.221 Z-7.000   ',
'G01 X-3.253 Y-13.080 Z-7.000   ',
'G01 X-3.895 Y-12.908 Z-7.000   ',
'G01 X-4.527 Y-12.705 Z-7.000   ',
'G01 X-5.149 Y-12.470 Z-7.000   ',
'G01 X-5.759 Y-12.206 Z-7.000   ',
'G01 X-6.355 Y-11.911 Z-7.000   ',
'G01 X-6.937 Y-11.588 Z-7.000   ',
'G01 X-7.502 Y-11.236 Z-7.000   ',
'G01 X-8.049 Y-10.857 Z-7.000   ',
'G01 X-8.577 Y-10.452 Z-7.000   ',
'G01 X-9.085 Y-10.020 Z-7.000   ',
'G01 X-9.572 Y-9.564 Z-7.000    ',
'G01 X-10.035 Y-9.085 Z-7.000   ',
'G01 X-10.475 Y-8.583 Z-7.000   ',
'G01 X-10.889 Y-8.060 Z-7.000   ',
'G01 X-11.278 Y-7.518 Z-7.000   ',
'G01 X-11.640 Y-6.956 Z-7.000   ',
'G01 X-11.974 Y-6.377 Z-7.000   ',
'G01 X-11.974 Y-6.377 Z-6.426   ',
'G01 X-12.279 Y-5.783 Z-6.426   ',
'G01 X-12.555 Y-5.174 Z-5.849   ',
'G01 X-12.800 Y-4.551 Z-5.554   ',
'G01 X-13.015 Y-3.918 Z-5.194   ',
'G01 X-13.199 Y-3.274 Z-4.941   ',
'G01 X-13.350 Y-2.622 Z-4.722   ',
'G01 X-13.470 Y-1.963 Z-4.620   ',
'G01 X-13.557 Y-1.298 Z-4.508   ',
'G01 X-13.612 Y-0.630 Z-4.464   ',
'G01 X-13.633 Y0.040 Z-4.510    ',
'G01 X-13.622 Y0.711 Z-4.466    ',
'G01 X-13.578 Y1.381 Z-4.517    ',
'G01 X-13.501 Y2.048 Z-4.636    ',
'G01 X-13.391 Y2.711 Z-4.743    ',
'G01 X-13.249 Y3.368 Z-4.974    ',
'G01 X-13.075 Y4.017 Z-5.236    ',
'G01 X-12.869 Y4.657 Z-5.609    ',
'G01 X-12.632 Y5.286 Z-6.111    ',
'G01 X-12.364 Y5.904 Z-6.536    ',
'G01 X-12.066 Y6.507 Z-6.536    ',
'G01 X-12.066 Y6.507 Z-7.000    ',
'G01 X-11.738 Y7.096 Z-7.000    ',
'G01 X-11.382 Y7.668 Z-7.000    ',
'G01 X-10.998 Y8.222 Z-7.000    ',
'G01 X-10.588 Y8.757 Z-7.000    ',
'G01 X-10.151 Y9.271 Z-7.000    ',
'G01 X-9.689 Y9.763 Z-7.000     ',
'G01 X-9.204 Y10.232 Z-7.000    ',
'G01 X-8.696 Y10.677 Z-7.000    ',
'G01 X-8.167 Y11.097 Z-7.000    ',
'G01 X-7.617 Y11.490 Z-7.000    ',
'G01 X-7.049 Y11.857 Z-7.000    ',
'G01 X-6.463 Y12.194 Z-7.000    ',
'G01 X-5.861 Y12.503 Z-7.000    ',
'G01 X-5.245 Y12.782 Z-7.000    ',
'G01 X-4.615 Y13.031 Z-7.000    ',
'G01 X-3.973 Y13.248 Z-7.000    ',
'G01 X-3.322 Y13.434 Z-7.000    ',
'G01 X-2.661 Y13.588 Z-7.000    ',
'G01 X-1.994 Y13.709 Z-7.000    ',
'G01 X-1.322 Y13.797 Z-7.000    ',
'G01 X-0.645 Y13.852 Z-7.000    ',
'G01 X0.033 Y13.874 Z-7.000     ',
'G01 X0.712 Y13.862 Z-7.000     ',
'G01 X1.390 Y13.818 Z-7.000     ',
'G01 X2.065 Y13.740 Z-7.000     ',
'G01 X2.736 Y13.628 Z-7.000     ',
'G01 X3.401 Y13.484 Z-7.000     ',
'G01 X4.058 Y13.308 Z-7.000     ',
'G01 X4.706 Y13.099 Z-7.000     ',
'G01 X4.706 Y13.099 Z-6.274     ',
'G01 X5.343 Y12.859 Z-6.274     ',
'G01 X5.343 Y12.859 Z-5.031     ',
'G01 X5.968 Y12.588 Z-5.031     ',
'G01 X6.579 Y12.286 Z-4.520     ',
'G01 X7.175 Y11.955 Z-4.064     ',
'G01 X7.175 Y11.955 Z-3.375     ',
'G01 X7.753 Y11.594 Z-3.375     ',
'G01 X8.314 Y11.206 Z-2.781     ',
'G01 X8.855 Y10.790 Z-2.258     ',
'G01 X9.376 Y10.348 Z-1.803     ',
'G01 X9.874 Y9.881 Z-1.411      ',
'G01 X10.349 Y9.390 Z-1.077     ',
'G01 X10.799 Y8.876 Z-0.791     ',
'G01 X11.224 Y8.340 Z-0.432     ',
'G01 X11.622 Y7.784 Z-0.300     ',
'G01 X11.992 Y7.208 Z-0.146     ',
'G01 X12.334 Y6.615 Z-0.075     ',
'G01 X12.647 Y6.006 Z-0.027     ',
'G01 X12.929 Y5.382 Z-0.002     ',
'G01 X13.181 Y4.745 Z0.000      ',
'G01 X13.401 Y4.095 Z0.000      ',
'G01 X13.589 Y3.436 Z0.000      ',
'G01 X13.744 Y2.768 Z0.000      ',
'G01 X13.866 Y2.092 Z0.000      ',
'G01 X13.956 Y1.412 Z0.000      ',
'G01 X14.011 Y0.727 Z0.000      ',
'G01 X14.033 Y0.040 Z0.000      ',
'G01 X14.023 Y-0.611 Z0.000     ',
'G01 X13.983 Y-1.262 Z0.000     ',
'G01 X13.912 Y-1.910 Z0.000     ',
'G01 X13.811 Y-2.555 Z0.000     ',
'G01 X13.680 Y-3.194 Z0.000     ',
'G01 X13.519 Y-3.827 Z0.000     ',
'G01 X13.330 Y-4.451 Z0.000     ',
'G01 X13.111 Y-5.067 Z0.000     ',
'G01 X12.864 Y-5.672 Z-0.016    ',
'G01 X12.588 Y-6.265 Z-0.024    ',
'G01 X12.286 Y-6.845 Z-0.101    ',
'G01 X11.956 Y-7.410 Z-0.262    ',
'G01 X11.601 Y-7.959 Z-0.363    ',
'G01 X11.220 Y-8.492 Z-0.512    ',
'G01 X10.815 Y-9.006 Z-0.952    ',
'G01 X10.386 Y-9.501 Z-1.238    ',
'G01 X9.934 Y-9.976 Z-1.576     ',
'G01 X9.461 Y-10.430 Z-1.950    ',
'G01 X8.966 Y-10.861 Z-2.418    ',
'G01 X8.453 Y-11.268 Z-2.962    ',
'G01 X7.920 Y-11.652 Z-3.582    ',
'G01 X7.370 Y-12.011 Z-3.927    ',
'G01 X6.804 Y-12.343 Z-3.927    ',
'G01 X6.804 Y-12.343 Z-4.738    ',
'G01 X6.222 Y-12.649 Z-5.261    ',
'G01 X5.627 Y-12.928 Z-5.261    ',
'G01 X5.627 Y-12.928 Z-5.970    ',
'G01 X5.020 Y-13.179 Z-5.970    ',
'G01 X5.020 Y-13.179 Z-6.928    ',
'G01 X4.401 Y-13.401 Z-6.928    ',
'G01 X4.401 Y-13.401 Z-7.000    ',
'G01 X3.772 Y-13.595 Z-7.000    ',
'G01 X3.135 Y-13.759 Z-7.000    ',
'G01 X2.490 Y-13.893 Z-7.000    ',
'G01 X1.840 Y-13.997 Z-7.000    ',
'G01 X1.185 Y-14.071 Z-7.000    ',
'G01 X0.528 Y-14.114 Z-7.000    ',
'G01 X-0.132 Y-14.126 Z-7.000   ',
'G01 X-0.791 Y-14.108 Z-7.000   ',
'G01 X-1.449 Y-14.060 Z-7.000   ',
'G01 X-2.104 Y-13.980 Z-7.000   ',
'G01 X-2.755 Y-13.871 Z-7.000   ',
'G01 X-3.400 Y-13.731 Z-7.000   ',
'G01 X-4.039 Y-13.561 Z-7.000   ',
'G01 X-4.669 Y-13.361 Z-7.000   ',
'G01 X-5.289 Y-13.132 Z-7.000   ',
'G01 X-5.898 Y-12.875 Z-7.000   ',
'G01 X-6.495 Y-12.589 Z-7.000   ',
'G01 X-7.078 Y-12.276 Z-7.000   ',
'G01 X-7.646 Y-11.936 Z-7.000   ',
'G01 X-8.198 Y-11.570 Z-7.000   ',
'G01 X-8.732 Y-11.178 Z-7.000   ',
'G01 X-9.248 Y-10.762 Z-7.000   ',
'G01 X-9.743 Y-10.322 Z-7.000   ',
'G01 X-10.219 Y-9.860 Z-7.000   ',
'G01 X-10.672 Y-9.375 Z-7.000   ',
'G01 X-11.102 Y-8.870 Z-7.000   ',
'G01 X-11.509 Y-8.345 Z-7.000   ',
'G01 X-11.890 Y-7.802 Z-7.000   ',
'G01 X-12.247 Y-7.241 Z-7.000   ',
'G01 X-12.576 Y-6.664 Z-7.000   ',
'G01 X-12.879 Y-6.072 Z-7.000   ',
'G01 X-12.879 Y-6.072 Z-6.343   ',
'G01 X-13.154 Y-5.467 Z-6.343   ',
'G01 X-13.401 Y-4.849 Z-5.816   ',
'G01 X-13.618 Y-4.220 Z-5.430   ',
'G01 X-13.807 Y-3.582 Z-5.158   ',
'G01 X-13.965 Y-2.935 Z-4.982   ',
'G01 X-14.093 Y-2.281 Z-4.843   ',
'G01 X-14.191 Y-1.622 Z-4.701   ',
'G01 X-14.258 Y-0.959 Z-4.631   ',
'G01 X-14.294 Y-0.293 Z-4.623   ',
'G01 X-14.299 Y0.374 Z-4.623    ',
'G01 X-14.272 Y1.041 Z-4.654    ',
'G01 X-14.215 Y1.706 Z-4.713    ',
'G01 X-14.127 Y2.368 Z-4.864    ',
'G01 X-14.009 Y3.025 Z-5.007    ',
'G01 X-13.859 Y3.676 Z-5.273    ',
'G01 X-13.680 Y4.320 Z-5.552    ',
'G01 X-13.470 Y4.955 Z-5.948    ',
'G01 X-13.232 Y5.580 Z-6.493    ',
'G01 X-12.964 Y6.194 Z-6.493    ',
'G01 X-12.964 Y6.194 Z-7.000    ',
'G01 X-12.668 Y6.794 Z-7.000    ',
'G01 X-12.344 Y7.380 Z-7.000    ',
'G01 X-11.994 Y7.951 Z-7.000    ',
'G01 X-11.617 Y8.505 Z-7.000    ',
'G01 X-11.214 Y9.040 Z-7.000    ',
'G01 X-10.787 Y9.557 Z-7.000    ',
'G01 X-10.336 Y10.054 Z-7.000   ',
'G01 X-9.862 Y10.529 Z-7.000    ',
'G01 X-9.367 Y10.982 Z-7.000    ',
'G01 X-8.850 Y11.411 Z-7.000    ',
'G01 X-8.315 Y11.816 Z-7.000    ',
'G01 X-7.760 Y12.196 Z-7.000    ',
'G01 X-7.189 Y12.550 Z-7.000    ',
'G01 X-6.601 Y12.877 Z-7.000    ',
'G01 X-5.999 Y13.176 Z-7.000    ',
'G01 X-5.383 Y13.447 Z-7.000    ',
'G01 X-4.755 Y13.689 Z-7.000    ',
'G01 X-4.116 Y13.902 Z-7.000    ',
'G01 X-3.468 Y14.085 Z-7.000    ',
'G01 X-2.812 Y14.237 Z-7.000    ',
'G01 X-2.149 Y14.359 Z-7.000    ',
'G01 X-1.481 Y14.450 Z-7.000    ',
'G01 X-0.809 Y14.510 Z-7.000    ',
'G01 X-0.135 Y14.538 Z-7.000    ',
'G01 X0.540 Y14.535 Z-7.000     ',
'G01 X1.214 Y14.501 Z-7.000     ',
'G01 X1.886 Y14.435 Z-7.000     ',
'G01 X2.554 Y14.338 Z-7.000     ',
'G01 X3.218 Y14.210 Z-7.000     ',
'G01 X3.875 Y14.052 Z-7.000     ',
'G01 X4.524 Y13.862 Z-7.000     ',
'G01 X5.164 Y13.643 Z-7.000     ',
'G01 X5.794 Y13.394 Z-7.000     ',
'G01 X5.794 Y13.394 Z-6.470     ',
'G01 X6.411 Y13.116 Z-6.470     ',
'G01 X6.411 Y13.116 Z-5.321     ',
'G01 X7.015 Y12.810 Z-5.321     ',
'G01 X7.604 Y12.475 Z-4.837     ',
'G01 X7.604 Y12.475 Z-4.052     ',
'G01 X8.177 Y12.114 Z-4.052     ',
'G01 X8.733 Y11.726 Z-3.700     ',
'G01 X9.270 Y11.312 Z-3.106     ',
'G01 X9.788 Y10.874 Z-2.592     ',
'G01 X10.285 Y10.412 Z-2.153    ',
'G01 X10.760 Y9.927 Z-1.564     ',
'G01 X11.212 Y9.420 Z-1.263     ',
'G01 X11.640 Y8.893 Z-1.015     ',
'G01 X12.043 Y8.346 Z-0.650     ',
'G01 X12.421 Y7.781 Z-0.515     ',
'G01 X12.772 Y7.199 Z-0.271     ',
'G01 X13.096 Y6.601 Z-0.232     ',
'G01 X13.391 Y5.988 Z-0.111     ',
'G01 X13.658 Y5.362 Z-0.042     ',
'G01 X13.896 Y4.724 Z-0.009     ',
'G01 X14.103 Y4.075 Z0.000      ',
'G01 X14.281 Y3.417 Z0.000      ',
'G01 X14.427 Y2.752 Z0.000      ',
'G01 X14.543 Y2.080 Z0.000      ',
'G01 X14.627 Y1.403 Z0.000      ',
'G01 X14.679 Y0.723 Z0.000      ',
'G01 X14.700 Y0.040 Z0.000      ',
'G01 X14.690 Y-0.613 Z0.000     ',
'G01 X14.651 Y-1.266 Z0.000     ',
'G01 X14.583 Y-1.916 Z0.000     ',
'G01 X14.486 Y-2.563 Z0.000     ',
'G01 X14.361 Y-3.206 Z0.000     ',
'G01 X14.206 Y-3.842 Z0.000     ',
'G01 X14.024 Y-4.471 Z-0.008    ',
'G01 X13.813 Y-5.091 Z-0.035    ',
'G01 X13.575 Y-5.702 Z-0.095    ',
'G01 X13.310 Y-6.301 Z-0.196    ',
'G01 X13.019 Y-6.889 Z-0.223    ',
'G01 X12.701 Y-7.463 Z-0.427    ',
'G01 X12.359 Y-8.022 Z-0.526    ',
'G01 X11.991 Y-8.566 Z-0.916    ',
'G01 X11.599 Y-9.093 Z-1.131    ',
'G01 X11.185 Y-9.602 Z-1.391    ',
'G01 X10.747 Y-10.093 Z-1.923   ',
'G01 X10.289 Y-10.563 Z-2.311   ',
'G01 X9.809 Y-11.013 Z-2.765    ',
'G01 X9.310 Y-11.442 Z-3.295    ',
'G01 X8.792 Y-11.847 Z-3.582    ',
'G01 X8.257 Y-12.229 Z-3.582    ',
'G01 X8.257 Y-12.229 Z-4.286    ',
'G01 X7.704 Y-12.588 Z-4.286    ',
'G01 X7.704 Y-12.588 Z-5.110    ',
'G01 X7.136 Y-12.921 Z-5.600    ',
'G01 X6.554 Y-13.229 Z-5.600    ',
'G01 X6.554 Y-13.229 Z-6.887    ',
'G01 X5.958 Y-13.510 Z-6.887    ',
'G01 X5.958 Y-13.510 Z-7.000    ',
'G01 X5.351 Y-13.765 Z-7.000    ',
'G01 X4.732 Y-13.993 Z-7.000    ',
'G01 X4.103 Y-14.193 Z-7.000    ',
'G01 X3.466 Y-14.365 Z-7.000    ',
'G01 X2.822 Y-14.508 Z-7.000    ',
'G01 X2.172 Y-14.622 Z-7.000    ',
'G01 X2.143 Y-14.626 Z-7.000    ',
'G00 X2.143 Y-14.626 Z2.000     ',
'G00 X-2.275 Y-14.626 Z2.000    ',
'G01 X-2.275 Y-14.626 Z-7.000   ',
'G01 X-2.437 Y-14.604 Z-7.000   ',
'G01 X-3.088 Y-14.484 Z-7.000   ',
'G01 X-3.733 Y-14.335 Z-7.000   ',
'G01 X-4.371 Y-14.157 Z-7.000   ',
'G01 X-5.001 Y-13.952 Z-7.000   ',
'G01 X-5.621 Y-13.718 Z-7.000   ',
'G01 X-6.230 Y-13.457 Z-7.000   ',
'G01 X-6.827 Y-13.168 Z-7.000   ',
'G01 X-7.411 Y-12.854 Z-7.000   ',
'G01 X-7.981 Y-12.513 Z-7.000   ',
'G01 X-8.535 Y-12.148 Z-7.000   ',
'G01 X-9.072 Y-11.758 Z-7.000   ',
'G01 X-9.592 Y-11.344 Z-7.000   ',
'G01 X-10.092 Y-10.907 Z-7.000  ',
'G01 X-10.573 Y-10.449 Z-7.000  ',
'G01 X-11.034 Y-9.969 Z-7.000   ',
'G01 X-11.472 Y-9.469 Z-7.000   ',
'G01 X-11.888 Y-8.950 Z-7.000   ',
'G01 X-12.281 Y-8.413 Z-7.000   ',
'G01 X-12.649 Y-7.858 Z-7.000   ',
'G01 X-12.992 Y-7.288 Z-7.000   ',
'G01 X-13.310 Y-6.702 Z-7.000   ',
'G01 X-13.602 Y-6.103 Z-7.000   ',
'G01 X-13.866 Y-5.491 Z-6.676   ',
'G01 X-14.103 Y-4.868 Z-6.155   ',
'G01 X-14.312 Y-4.235 Z-5.785   ',
'G01 X-14.493 Y-3.593 Z-5.418   ',
'G01 X-14.645 Y-2.943 Z-5.225   ',
'G01 X-14.768 Y-2.287 Z-5.091   ',
'G01 X-14.862 Y-1.626 Z-4.943   ',
'G01 X-14.926 Y-0.961 Z-4.885   ',
'G01 X-14.961 Y-0.294 Z-4.863   ',
'G01 X-14.965 Y0.375 Z-4.863    ',
'G01 X-14.940 Y1.043 Z-4.892    ',
'G01 X-14.885 Y1.709 Z-5.000    ',
'G01 X-14.801 Y2.373 Z-5.114    ',
'G01 X-14.687 Y3.032 Z-5.260    ',
'G01 X-14.544 Y3.686 Z-5.569    ',
'G01 X-14.371 Y4.333 Z-5.835    ',
'G01 X-14.170 Y4.972 Z-6.225    ',
'G01 X-13.941 Y5.602 Z-6.769    ',
'G01 X-13.683 Y6.221 Z-6.769    ',
'G01 X-13.683 Y6.221 Z-7.000    ',
'G01 X-13.399 Y6.828 Z-7.000    ',
'G01 X-13.087 Y7.422 Z-7.000    ',
'G01 X-12.749 Y8.002 Z-7.000    ',
'G01 X-12.386 Y8.566 Z-7.000    ',
'G01 X-11.998 Y9.113 Z-7.000    ',
'G01 X-11.585 Y9.643 Z-7.000    ',
'G01 X-11.149 Y10.155 Z-7.000   ',
'G01 X-10.691 Y10.646 Z-7.000   ',
'G01 X-10.211 Y11.117 Z-7.000   ',
'G01 X-9.711 Y11.566 Z-7.000    ',
'G01 X-9.190 Y11.992 Z-7.000    ',
'G01 X-8.652 Y12.395 Z-7.000    ',
'G01 X-8.095 Y12.774 Z-7.000    ',
'G01 X-7.522 Y13.127 Z-7.000    ',
'G01 X-6.934 Y13.455 Z-7.000    ',
'G01 X-6.331 Y13.756 Z-7.000    ',
'G01 X-5.716 Y14.030 Z-7.000    ',
'G01 X-5.089 Y14.277 Z-7.000    ',
'G01 X-4.451 Y14.496 Z-7.000    ',
'G01 X-3.804 Y14.686 Z-7.000    ',
'G01 X-3.716 Y14.707 Z-7.000    ',
'G00 X-3.716 Y14.707 Z2.000     ',
'G00 X3.991 Y14.707 Z2.000      ',
'G01 X3.991 Y14.707 Z-7.000     ',
'G01 X4.211 Y14.651 Z-7.000     ',
'G01 X4.859 Y14.455 Z-7.000     ',
'G01 X5.498 Y14.230 Z-7.000     ',
'G01 X6.127 Y13.977 Z-7.000     ',
'G01 X6.744 Y13.696 Z-7.000     ',
'G01 X6.744 Y13.696 Z-7.000     ',
'G01 X7.348 Y13.388 Z-7.000     ',
'G01 X7.937 Y13.052 Z-6.338     ',
'G01 X7.937 Y13.052 Z-5.281     ',
'G01 X8.512 Y12.691 Z-5.281     ',
'G01 X8.512 Y12.691 Z-4.449     ',
'G01 X9.070 Y12.305 Z-4.449     ',
'G01 X9.070 Y12.305 Z-3.762     ',
'G01 X9.610 Y11.894 Z-3.762     ',
'G01 X10.132 Y11.459 Z-3.193    ',
'G01 X10.634 Y11.001 Z-2.766    ',
'G01 X11.115 Y10.521 Z-2.364    ',
'G01 X11.574 Y10.020 Z-2.026    ',
'G01 X12.011 Y9.499 Z-1.746     ',
'G01 X12.425 Y8.959 Z-1.324     ',
'G01 X12.814 Y8.401 Z-1.157     ',
'G01 X13.177 Y7.826 Z-0.770     ',
'G01 X13.515 Y7.235 Z-0.562     ',
'G01 X13.827 Y6.629 Z-0.439     ',
'G01 X14.111 Y6.010 Z-0.273     ',
'G01 X14.367 Y5.378 Z-0.215     ',
'G01 X14.595 Y4.736 Z-0.131     ',
'G01 X14.794 Y4.084 Z-0.044     ',
'G01 X14.965 Y3.423 Z-0.028     ',
'G01 X15.105 Y2.756 Z-0.021     ',
'G01 X15.216 Y2.082 Z-0.007     ',
'G01 X15.296 Y1.404 Z-0.011     ',
'G01 X15.347 Y0.723 Z-0.008     ',
'G01 X15.367 Y0.040 Z-0.008     ',
'G01 X15.357 Y-0.615 Z-0.008    ',
'G01 X15.320 Y-1.270 Z-0.010    ',
'G01 X15.254 Y-1.922 Z-0.006    ',
'G01 X15.161 Y-2.571 Z-0.018    ',
'G01 X15.040 Y-3.216 Z-0.052    ',
'G01 X14.892 Y-3.856 Z-0.075    ',
'G01 X14.716 Y-4.488 Z-0.085    ',
'G01 X14.513 Y-5.113 Z-0.147    ',
'G01 X14.284 Y-5.729 Z-0.250    ',
'G01 X14.028 Y-6.334 Z-0.399    ',
'G01 X13.747 Y-6.929 Z-0.503    ',
'G01 X13.441 Y-7.511 Z-0.672    ',
'G01 X13.110 Y-8.079 Z-1.027    ',
'G01 X12.755 Y-8.633 Z-1.172    ',
'G01 X12.376 Y-9.171 Z-1.447    ',
'G01 X11.975 Y-9.693 Z-1.884    ',
'G01 X11.551 Y-10.198 Z-2.175   ',
'G01 X11.107 Y-10.683 Z-2.525   ',
'G01 X10.641 Y-11.150 Z-2.942   ',
'G01 X10.157 Y-11.597 Z-3.436   ',
'G01 X9.653 Y-12.022 Z-3.987    ',
'G01 X9.131 Y-12.426 Z-3.987    ',
'G01 X9.131 Y-12.426 Z-4.701    ',
'G01 X8.593 Y-12.807 Z-4.701    ',
'G01 X8.593 Y-12.807 Z-5.586    ',
'G01 X8.038 Y-13.165 Z-6.118    ',
'G01 X7.469 Y-13.499 Z-6.118    ',
'G01 X7.469 Y-13.499 Z-7.000    ',
'G01 X6.886 Y-13.808 Z-7.000    ',
'G01 X6.290 Y-14.093 Z-7.000    ',
'G01 X5.682 Y-14.351 Z-7.000    ',
'G01 X5.063 Y-14.584 Z-7.000    ',
'G01 X4.933 Y-14.626 Z-7.000    ',
'G00 X4.933 Y-14.626 Z2.000     ',
'G00 X-5.079 Y-14.626 Z2.000    ',
'G01 X-5.079 Y-14.626 Z-7.000   ',
'G01 X-5.333 Y-14.541 Z-7.000   ',
'G01 X-5.953 Y-14.302 Z-7.000   ',
'G01 X-6.562 Y-14.038 Z-7.000   ',
'G01 X-7.160 Y-13.747 Z-7.000   ',
'G01 X-7.744 Y-13.431 Z-7.000   ',
'G01 X-8.315 Y-13.090 Z-7.000   ',
'G01 X-8.871 Y-12.725 Z-7.000   ',
'G01 X-9.412 Y-12.337 Z-7.000   ',
'G01 X-9.935 Y-11.925 Z-7.000   ',
'G01 X-10.440 Y-11.492 Z-7.000  ',
'G01 X-10.926 Y-11.037 Z-7.000  ',
'G01 X-11.393 Y-10.562 Z-7.000  ',
'G01 X-11.839 Y-10.067 Z-7.000  ',
'G01 X-12.264 Y-9.553 Z-7.000   ',
'G01 X-12.666 Y-9.021 Z-7.000   ',
'G01 X-13.045 Y-8.473 Z-7.000   ',
'G01 X-13.401 Y-7.909 Z-7.000   ',
'G01 X-13.733 Y-7.329 Z-7.000   ',
'G01 X-14.039 Y-6.736 Z-7.000   ',
'G01 X-14.320 Y-6.131 Z-7.000   ',
'G01 X-14.575 Y-5.513 Z-7.000   ',
'G01 X-14.803 Y-4.886 Z-6.548   ',
'G01 X-15.004 Y-4.248 Z-6.175   ',
'G01 X-15.178 Y-3.603 Z-5.764   ',
'G01 X-15.324 Y-2.950 Z-5.549   ',
'G01 X-15.443 Y-2.292 Z-5.429   ',
'G01 X-15.533 Y-1.629 Z-5.317   ',
'G01 X-15.594 Y-0.963 Z-5.214   ',
'G01 X-15.627 Y-0.294 Z-5.191   ',
'G01 X-15.632 Y0.375 Z-5.191    ',
'G01 X-15.608 Y1.045 Z-5.221    ',
'G01 X-15.555 Y1.713 Z-5.336    ',
'G01 X-15.474 Y2.378 Z-5.533    ',
'G01 X-15.364 Y3.039 Z-5.584    ',
'G01 X-15.227 Y3.695 Z-5.941    ',
'G01 X-15.061 Y4.345 Z-6.233    ',
'G01 X-14.867 Y4.988 Z-6.620    ',
'G01 X-14.647 Y5.622 Z-7.000    ',
'G01 X-14.399 Y6.246 Z-7.000    ',
'G01 X-14.125 Y6.859 Z-7.000    ',
'G01 X-13.824 Y7.460 Z-7.000    ',
'G01 X-13.499 Y8.047 Z-7.000    ',
'G01 X-13.148 Y8.621 Z-7.000    ',
'G01 X-12.773 Y9.179 Z-7.000    ',
'G01 X-12.374 Y9.720 Z-7.000    ',
'G01 X-11.953 Y10.245 Z-7.000   ',
'G01 X-11.509 Y10.750 Z-7.000   ',
'G01 X-11.044 Y11.237 Z-7.000   ',
'G01 X-10.559 Y11.704 Z-7.000   ',
'G01 X-10.054 Y12.149 Z-7.000   ',
'G01 X-9.530 Y12.573 Z-7.000    ',
'G01 X-8.988 Y12.974 Z-7.000    ',
'G01 X-8.430 Y13.351 Z-7.000    ',
'G01 X-7.856 Y13.704 Z-7.000    ',
'G01 X-7.267 Y14.033 Z-7.000    ',
'G01 X-6.664 Y14.336 Z-7.000    ',
'G01 X-6.049 Y14.614 Z-7.000    ',
'G01 X-5.815 Y14.707 Z-7.000    ',
'G00 X-5.815 Y14.707 Z2.000     ',
'G00 X6.099 Y14.707 Z2.000      ',
'G01 X6.099 Y14.707 Z-7.000     ',
'G01 X6.460 Y14.559 Z-7.000     ',
'G01 X7.077 Y14.275 Z-7.000     ',
'G01 X7.681 Y13.965 Z-7.000     ',
'G01 X8.271 Y13.630 Z-7.000     ',
'G01 X8.847 Y13.269 Z-7.000     ',
'G01 X8.847 Y13.269 Z-5.830     ',
'G01 X9.407 Y12.884 Z-5.830     ',
'G01 X9.407 Y12.884 Z-4.999     ',
'G01 X9.950 Y12.475 Z-4.999     ',
'G01 X9.950 Y12.475 Z-4.303     ',
'G01 X10.475 Y12.044 Z-4.303    ',
'G01 X10.982 Y11.590 Z-3.727    ',
'G01 X11.468 Y11.115 Z-3.249    ',
'G01 X11.934 Y10.619 Z-2.944    ',
'G01 X12.379 Y10.104 Z-2.376    ',
'G01 X12.801 Y9.570 Z-2.022     ',
'G01 X13.201 Y9.018 Z-1.620     ',
'G01 X13.576 Y8.449 Z-1.479     ',
'G01 X13.927 Y7.865 Z-1.217     ',
'G01 X14.253 Y7.266 Z-1.040     ',
'G01 X14.553 Y6.654 Z-0.762     ',
'G01 X14.826 Y6.029 Z-0.643     ',
'G01 X15.073 Y5.393 Z-0.463     ',
'G01 X15.292 Y4.747 Z-0.346     ',
'G01 X15.484 Y4.092 Z-0.272     ',
'G01 X15.647 Y3.429 Z-0.163     ',
'G01 X15.782 Y2.760 Z-0.155     ',
'G01 X15.888 Y2.085 Z-0.103     ',
'G01 X15.966 Y1.406 Z-0.135     ',
'G01 X16.014 Y0.724 Z-0.121     ',
'G01 X16.033 Y0.040 Z-0.120     ',
'G01 X16.024 Y-0.617 Z-0.121    ',
'G01 X15.988 Y-1.273 Z-0.132    ',
'G01 X15.925 Y-1.927 Z-0.162    ',
'G01 X15.835 Y-2.579 Z-0.147    ',
'G01 X15.719 Y-3.226 Z-0.226    ',
'G01 X15.575 Y-3.869 Z-0.257    ',
'G01 X15.406 Y-4.505 Z-0.268    ',
'G01 X15.211 Y-5.133 Z-0.359    ',
'G01 X14.989 Y-5.754 Z-0.501    ',
'G01 X14.743 Y-6.364 Z-0.716    ',
'G01 X14.472 Y-6.965 Z-0.976    ',
'G01 X14.176 Y-7.554 Z-1.135    ',
'G01 X13.856 Y-8.130 Z-1.361    ',
'G01 X13.512 Y-8.693 Z-1.593    ',
'G01 X13.146 Y-9.242 Z-1.948    ',
'G01 X12.757 Y-9.775 Z-2.163    ',
'G01 X12.347 Y-10.292 Z-2.429   ',
'G01 X11.915 Y-10.792 Z-3.029   ',
'G01 X11.464 Y-11.273 Z-3.445   ',
'G01 X10.993 Y-11.736 Z-3.947   ',
'G01 X10.503 Y-12.180 Z-4.549   ',
'G01 X9.995 Y-12.602 Z-4.549    ',
'G01 X9.995 Y-12.602 Z-5.286    ',
'G01 X9.470 Y-13.004 Z-5.286    ',
'G01 X9.470 Y-13.004 Z-6.176    ',
'G01 X8.929 Y-13.384 Z-6.751    ',
'G01 X8.373 Y-13.742 Z-6.751    ',
'G01 X8.373 Y-13.742 Z-7.000    ',
'G01 X7.802 Y-14.077 Z-7.000    ',
'G01 X7.218 Y-14.387 Z-7.000    ',
'G01 X6.721 Y-14.626 Z-7.000    ',
'G00 X6.721 Y-14.626 Z2.000     ',
'G00 X-6.877 Y-14.626 Z2.000    ',
'G01 X-6.877 Y-14.626 Z-7.000   ',
'G01 X-6.894 Y-14.619 Z-7.000   ',
'G01 X-7.492 Y-14.326 Z-7.000   ',
'G01 X-8.078 Y-14.008 Z-7.000   ',
'G01 X-8.650 Y-13.667 Z-7.000   ',
'G01 X-9.208 Y-13.303 Z-7.000   ',
'G01 X-9.751 Y-12.916 Z-7.000   ',
'G01 X-10.277 Y-12.506 Z-7.000  ',
'G01 X-10.786 Y-12.076 Z-7.000  ',
'G01 X-11.278 Y-11.624 Z-7.000  ',
'G01 X-11.750 Y-11.153 Z-7.000  ',
'G01 X-12.203 Y-10.663 Z-7.000  ',
'G01 X-12.636 Y-10.154 Z-7.000  ',
'G01 X-13.047 Y-9.628 Z-7.000   ',
'G01 X-13.437 Y-9.085 Z-7.000   ',
'G01 X-13.804 Y-8.527 Z-7.000   ',
'G01 X-14.147 Y-7.954 Z-7.000   ',
'G01 X-14.468 Y-7.367 Z-7.000   ',
'G01 X-14.763 Y-6.767 Z-7.000   ',
'G01 X-15.034 Y-6.156 Z-7.000   ',
'G01 X-15.280 Y-5.533 Z-7.000   ',
'G01 X-15.500 Y-4.901 Z-7.000   ',
'G01 X-15.694 Y-4.260 Z-6.682   ',
'G01 X-15.862 Y-3.612 Z-6.356   ',
'G01 X-16.003 Y-2.957 Z-5.983   ',
'G01 X-16.116 Y-2.297 Z-5.964   ',
'G01 X-16.203 Y-1.632 Z-5.760   ',
'G01 X-16.262 Y-0.965 Z-5.648   ',
'G01 X-16.294 Y-0.295 Z-5.621   ',
'G01 X-16.299 Y0.376 Z-5.621    ',
'G01 X-16.276 Y1.046 Z-5.657    ',
'G01 X-16.225 Y1.716 Z-5.781    ',
'G01 X-16.147 Y2.382 Z-5.995    ',
'G01 X-16.041 Y3.045 Z-6.135    ',
'G01 X-15.908 Y3.704 Z-6.409    ',
'G01 X-15.749 Y4.356 Z-6.752    ',
'G01 X-15.563 Y5.002 Z-7.000    ',
'G01 X-15.350 Y5.639 Z-7.000    ',
'G01 X-15.111 Y6.268 Z-7.000    ',
'G01 X-14.846 Y6.886 Z-7.000    ',
'G01 X-14.557 Y7.493 Z-7.000    ',
'G01 X-14.242 Y8.088 Z-7.000    ',
'G01 X-13.904 Y8.670 Z-7.000    ',
'G01 X-13.541 Y9.237 Z-7.000    ',
'G01 X-13.156 Y9.789 Z-7.000    ',
'G01 X-12.748 Y10.325 Z-7.000   ',
'G01 X-12.318 Y10.844 Z-7.000   ',
'G01 X-11.867 Y11.345 Z-7.000   ',
'G01 X-11.396 Y11.827 Z-7.000   ',
'G01 X-10.905 Y12.290 Z-7.000   ',
'G01 X-10.396 Y12.732 Z-7.000   ',
'G01 X-9.869 Y13.153 Z-7.000    ',
'G01 X-9.325 Y13.552 Z-7.000    ',
'G01 X-8.764 Y13.929 Z-7.000    ',
'G01 X-8.189 Y14.282 Z-7.000    ',
'G01 X-7.599 Y14.611 Z-7.000    ',
'G01 X-7.410 Y14.707 Z-7.000    ',
'G00 X-7.410 Y14.707 Z2.000     ',
'G00 X7.696 Y14.707 Z2.000      ',
'G01 X7.696 Y14.707 Z-7.000     ',
'G01 X8.014 Y14.543 Z-7.000     ',
'G01 X8.605 Y14.207 Z-7.000     ',
'G01 X9.182 Y13.847 Z-7.000     ',
'G01 X9.743 Y13.463 Z-7.000     ',
'G01 X10.289 Y13.056 Z-6.625    ',
'G01 X10.289 Y13.056 Z-5.769    ',
'G01 X10.817 Y12.628 Z-5.769    ',
'G01 X10.817 Y12.628 Z-5.032    ',
'G01 X11.328 Y12.178 Z-5.032    ',
'G01 X11.328 Y12.178 Z-4.079    ',
'G01 X11.820 Y11.707 Z-4.079    ',
'G01 X12.292 Y11.216 Z-3.631    ',
'G01 X12.744 Y10.706 Z-3.263    ',
'G01 X13.175 Y10.178 Z-2.965    ',
'G01 X13.583 Y9.632 Z-2.486     ',
'G01 X13.969 Y9.070 Z-2.319     ',
'G01 X14.332 Y8.493 Z-1.863     ',
'G01 X14.671 Y7.901 Z-1.621     ',
'G01 X14.985 Y7.295 Z-1.455     ',
'G01 X15.274 Y6.677 Z-1.303     ',
'G01 X15.538 Y6.047 Z-1.052     ',
'G01 X15.776 Y5.407 Z-0.851     ',
'G01 X15.987 Y4.757 Z-0.703     ',
'G01 X16.171 Y4.099 Z-0.614     ',
'G01 X16.329 Y3.434 Z-0.440     ',
'G01 X16.458 Y2.763 Z-0.437     ',
'G01 X16.561 Y2.087 Z-0.350     ',
'G01 X16.635 Y1.407 Z-0.412     ',
'G01 X16.682 Y0.725 Z-0.388     ',
'G01 X16.700 Y0.040 Z-0.386     ',
'G01 X16.691 Y-0.614 Z-0.387    ',
'G01 X16.657 Y-1.268 Z-0.406    ',
'G01 X16.597 Y-1.920 Z-0.463    ',
'G01 X16.511 Y-2.569 Z-0.424    ',
'G01 X16.400 Y-3.215 Z-0.550    ',
'G01 X16.264 Y-3.856 Z-0.588    ',
'G01 X16.102 Y-4.491 Z-0.594    ',
'G01 X15.916 Y-5.120 Z-0.710    ',
'G01 X15.705 Y-5.741 Z-1.036    ',
'G01 X15.470 Y-6.354 Z-1.119    ',
'G01 X15.211 Y-6.956 Z-1.252    ',
'G01 X14.928 Y-7.549 Z-1.551    ',
'G01 X14.622 Y-8.130 Z-1.904    ',
'G01 X14.294 Y-8.698 Z-1.980    ',
'G01 X13.943 Y-9.254 Z-2.454    ',
'G01 X13.571 Y-9.795 Z-2.636    ',
'G01 X13.178 Y-10.322 Z-3.136   ',
'G01 X12.764 Y-10.832 Z-3.449   ',
'G01 X12.330 Y-11.327 Z-3.835   ',
'G01 X11.877 Y-11.804 Z-4.306   ',
'G01 X11.406 Y-12.263 Z-4.880   ',
'G01 X10.917 Y-12.703 Z-4.880   ',
'G01 X10.917 Y-12.703 Z-5.583   ',
'G01 X10.411 Y-13.123 Z-5.583   ',
'G01 X10.411 Y-13.123 Z-6.495   ',
'G01 X9.889 Y-13.524 Z-6.495    ',
'G01 X9.889 Y-13.524 Z-7.000    ',
'G01 X9.351 Y-13.904 Z-7.000    ',
'G01 X8.798 Y-14.263 Z-7.000    ',
'G01 X8.232 Y-14.599 Z-7.000    ',
'G01 X8.182 Y-14.626 Z-7.000    ',
'G00 X8.182 Y-14.626 Z2.000     ',
'G00 X-8.335 Y-14.626 Z2.000    ',
'G01 X-8.335 Y-14.626 Z-7.000   ',
'G01 X-8.793 Y-14.362 Z-7.000   ',
'G01 X-9.353 Y-14.008 Z-7.000   ',
'G01 X-9.900 Y-13.632 Z-7.000   ',
'G01 X-10.432 Y-13.235 Z-7.000  ',
'G01 X-10.948 Y-12.817 Z-7.000  ',
'G01 X-11.447 Y-12.379 Z-7.000  ',
'G01 X-11.929 Y-11.921 Z-7.000  ',
'G01 X-12.392 Y-11.445 Z-7.000  ',
'G01 X-12.837 Y-10.951 Z-7.000  ',
'G01 X-13.261 Y-10.440 Z-7.000  ',
'G01 X-13.666 Y-9.913 Z-7.000   ',
'G01 X-14.050 Y-9.370 Z-7.000   ',
'G01 X-14.412 Y-8.812 Z-7.000   ',
'G01 X-14.752 Y-8.240 Z-7.000   ',
'G01 X-15.069 Y-7.655 Z-7.000   ',
'G01 X-15.363 Y-7.058 Z-7.000   ',
'G01 X-15.634 Y-6.449 Z-7.000   ',
'G01 X-15.881 Y-5.831 Z-7.000   ',
'G01 X-16.103 Y-5.203 Z-7.000   ',
'G01 X-16.300 Y-4.566 Z-7.000   ',
'G01 X-16.473 Y-3.922 Z-7.000   ',
'G01 X-16.620 Y-3.272 Z-6.833   ',
'G01 X-16.741 Y-2.616 Z-6.449   ',
'G01 X-16.836 Y-1.956 Z-6.405   ',
'G01 X-16.906 Y-1.293 Z-6.250   ',
'G01 X-16.949 Y-0.627 Z-6.191   ',
'G01 X-16.967 Y0.040 Z-6.189    ',
'G01 X-16.958 Y0.708 Z-6.194    ',
'G01 X-16.923 Y1.375 Z-6.263    ',
'G01 X-16.861 Y2.040 Z-6.434    ',
'G01 X-16.774 Y2.702 Z-6.719    ',
'G01 X-16.660 Y3.361 Z-6.887    ',
'G01 X-16.521 Y4.015 Z-7.000    ',
'G01 X-16.356 Y4.663 Z-7.000    ',
'G01 X-16.166 Y5.304 Z-7.000    ',
'G01 X-15.951 Y5.937 Z-7.000    ',
'G01 X-15.711 Y6.562 Z-7.000    ',
'G01 X-15.447 Y7.177 Z-7.000    ',
'G01 X-15.158 Y7.781 Z-7.000    ',
'G01 X-14.846 Y8.373 Z-7.000    ',
'G01 X-14.511 Y8.953 Z-7.000    ',
'G01 X-14.154 Y9.520 Z-7.000    ',
'G01 X-13.774 Y10.072 Z-7.000   ',
'G01 X-13.373 Y10.609 Z-7.000   ',
'G01 X-12.951 Y11.130 Z-7.000   ',
'G01 X-12.508 Y11.634 Z-7.000   ',
'G01 X-12.046 Y12.120 Z-7.000   ',
'G01 X-11.566 Y12.588 Z-7.000   ',
'G01 X-11.067 Y13.037 Z-7.000   ',
'G01 X-10.551 Y13.466 Z-7.000   ',
'G01 X-10.018 Y13.875 Z-7.000   ',
'G01 X-9.469 Y14.262 Z-7.000    ',
'G01 X-8.906 Y14.628 Z-7.000    ',
'G01 X-8.772 Y14.707 Z-7.000    ',
'G00 X-8.772 Y14.707 Z2.000     ',
'G00 X9.065 Y14.707 Z2.000      ',
'G01 X9.065 Y14.707 Z-7.000     ',
'G01 X9.605 Y14.366 Z-7.000     ',
'G01 X10.163 Y13.983 Z-7.000    ',
'G01 X10.705 Y13.577 Z-7.000    ',
'G01 X11.231 Y13.151 Z-7.000    ',
'G01 X11.231 Y13.151 Z-6.265    ',
'G01 X11.740 Y12.704 Z-6.265    ',
'G01 X11.740 Y12.704 Z-5.535    ',
'G01 X12.231 Y12.238 Z-5.535    ',
'G01 X12.703 Y11.753 Z-4.964    ',
'G01 X12.703 Y11.753 Z-4.149    ',
'G01 X13.157 Y11.249 Z-4.149    ',
'G01 X13.590 Y10.728 Z-3.809    ',
'G01 X14.002 Y10.190 Z-3.545    ',
'G01 X14.394 Y9.636 Z-3.082     ',
'G01 X14.763 Y9.067 Z-2.777     ',
'G01 X15.109 Y8.483 Z-2.479		'			
	];

	programmed_velocity: LREAL;
	state: sc_enum_program_status;
	mdi: STRING;
	mdi_start: BOOL;
	x_up: BOOL;
	x_dn: BOOL;
	y_up: BOOL;
	y_dn: BOOL;
	z_up: BOOL;
	z_dn: BOOL;
	optimizer: BOOL;
END_VAR
VAR // added by the converter: edge detectors and wires of the graphical bodies
    _s1 : cn_jog_cmd;
    _s2 : cn_limits;
END_VAR

// compose _s1 : cn_jog_cmd
_s1.jog_enable := jog_enable;
_s1.x_up := x_up;
_s1.x_dn := x_dn;
_s1.y_up := y_up;
_s1.y_dn := y_dn;
_s1.z_up := z_up;
_s1.z_dp := z_dn;
cnc_0(
    limits := _s2,
    jog_cmd := _s1,
    start := start,
    stop := stop,
    pause := pause,
    feed_override := feed_override,
    start_line := start_line,
    gcode_lines := gcode,
    mdi_line := mdi,
    mdi_start := mdi_start); // cnc
// compose _s2 : cn_limits
_s2.max_vel := maxvel;
_s2.max_acc := maxacc;
_s2.max_jerk := maxjerk;
_s2.max_quote_x := 250;
_s2.min_quote_x := -10;
_s2.max_quote_y := 250;
_s2.min_quote_y := -10;
_s2.max_quote_z := 20;
_s2.min_quote_z := -20;
line_nr := cnc_0.line_nr;
x := cnc_0.xyz.sc_pnt;
velocity := cnc_0.velocity;
y := cnc_0.xyz.x;
acceleration := cnc_0.acceleration;
programmed_velocity := cnc_0.programmed_velocity;
z := cnc_0.xyz.y;
line_progress := cnc_0.line_progress;
state := cnc_0.state;
performance := cnc_0.performance_msec;

END_PROGRAM

// MyController/Application/cnc/cnc
FUNCTION_BLOCK cnc
VAR_INPUT
	limits:cn_limits;
	jog_cmd:cn_jog_cmd;
	start:BOOL;
	stop:BOOL;
	pause:BOOL;
	feed_override:LREAL;
	start_line:UDINT;
	gcode_lines:REFERENCE TO ARRAY[0..MAX_GCODE_LINE]OF STRING(250);
	mdi_line:REFERENCE TO STRING(250);
	mdi_start:BOOL;
END_VAR
VAR_OUTPUT
	line_nr:UDINT;
	finished:BOOL;
	xyz:sc_pnt;
	velocity:LREAL;
	programmed_velocity:LREAL;
	acceleration:LREAL;
	line_progress:LREAL;	
	state:sc_enum_program_status:=program_end;
	performance_msec:LREAL;
END_VAR
VAR
	motion:sc_engine;
	motion_data:sc_data;
	motion_vec:vector_sc_segment;	//buffer vector to engine	
	parsed_vec:vector_sc_segment;   //buffer vector from gcode parser
	plv:sc_segment;
	error_on_line:UDINT;	
	syntax_error:BOOL;
	
	maxvel_fo:LREAL;
	maxvel_fo_old:LREAL;
	maxvel_foo:LREAL;

	engine_finished:BOOL;
	engine_fwd:BOOL;
	engine_rev:BOOL;
	engine_tarpos:LREAL;
	engine_endvel:LREAL;	
	engine_outpos:LREAL;
	stop_tarpos:LREAL;
	p:sc_segment;	
	t1,t2:ULINT;
	cycle_time:LREAL;
	upStart:R_TRIG;
	upStop:R_TRIG;
	upPause:R_TRIG;
	dnPause:F_TRIG;
	upJogEnable:R_TRIG;
	upMdiStart:R_TRIG;
	a,dv,gforcemax:LREAL;//optimizer
	line_nr_old:UDINT;
	stop_request:BOOL;
	pause_request:BOOL;
	resume_request:BOOL;
	set_start_on_current_position:BOOL;
	i,ii:UDINT;
	
	//jog
	jog_ovr:LREAL;
	jog_pos:LREAL;
	upJogPlus:R_TRIG;
	upJogMin:R_TRIG;
	dnJogPlusMin:F_TRIG;
	jog_tarpos:LREAL;
	jog_vel:LREAL;
END_VAR

//get time cycle from plc
SysTimeGetUs(t1);
cycle_time:=ULINT_TO_LREAL(t1-t2)/1000000;
t2:=t1;
performance_msec:=cycle_time;

//get data from current vector
p:=vector_at(motion_vec,line_nr);

//update motion 
update_motion_and_interpolator();

//optimizer on fly
IF(line_nr<>line_nr_old)THEN
	sc_optimize_all(motion_vec,line_nr,line_nr+MAX_LOOK_HEAD_LINE);
	line_nr_old:=line_nr;
END_IF

//jog
upJogEnable(CLK:=jog_cmd.jog_enable);
IF(jog_cmd.jog_enable AND state=program_end)THEN
	motion.set_pos(0,motion_data);	
	state:=program_jog;
END_IF

//mdi
upMdiStart(CLK:=mdi_start);
IF(upMdiStart.Q AND state=program_end)THEN
	sc_parse_clean();
	set_start_on_current_position:=TRUE;
	sc_parse_line(mdi_line);		
	motion_vec.clear();		
	motion_vec.insert(0,parsed_vec);
	motion.set_pos(0,motion_data);	
	state:=program_run;
END_IF

//start
upStart(CLK:=start);
IF(upStart.Q AND state=program_end)THEN
	state:=program_start;
END_IF

//stop
upStop(CLK:=stop);
IF(upStop.Q AND state=program_run)THEN
	stop_request:=TRUE;
END_IF

//pause
upPause(CLK:=pause);
IF(upPause.Q AND state=program_run)THEN
	pause_request:=TRUE;
END_IF

//pause resume
dnPause(CLK:=pause);
IF(dnPause.Q AND state=program_pause)THEN
	resume_request:=TRUE;
END_IF

//program state
CASE state OF
	program_start://-------------------------------------------------------------------------------------------
	
		line_nr:=start_line;
		sc_parse_clean();
		set_start_on_current_position:=TRUE;		
		sc_parse_start();		
		motion_vec.clear();		
		motion_vec.insert(0,parsed_vec);
		motion.set_pos(0,motion_data);	
		sc_optimize_all(motion_vec,0,MAX_LOOK_HEAD_LINE);			
		state:=program_run;	
	
	program_run://-------------------------------------------------------------------------------------------
	
		finished:=FALSE;	
		//line increment
		IF(engine_finished)THEN
			//cycle vectors			
			IF(motion_vec.data[line_nr+1].path_lenght=0)THEN
				IF(motion_vec.data[line_nr+1].primitive_id <> sc_primitive_id.empty)THEN
					WHILE motion_vec.data[line_nr+1].path_lenght=0 DO 
						IF(line_nr+1=motion_vec.size())THEN
							EXIT;
						END_IF
						vector_nr_increment(motion_vec,line_nr);
					END_WHILE
				ELSE
					vector_nr_increment(motion_vec,line_nr);
				END_IF
			ELSE
				vector_nr_increment(motion_vec,line_nr);				
			END_IF								
		END_IF
				
		IF(velocity=0)THEN
			IF(pause_request)THEN
				pause_request:=FALSE;
				state:=program_pause;
			END_IF
			IF(stop_request)THEN
				stop_request:=FALSE;
				state:=program_stop;
			END_IF
		END_IF
		
		//end program
		IF(engine_finished AND line_nr=motion_vec.size())THEN
			state:=program_end;
		END_IF
		
	program_pause://-------------------------------------------------------------------------------------------
	
		IF(resume_request)THEN
			resume_request:=FALSE;
			state:=program_run;
		END_IF
			
	program_stop://-------------------------------------------------------------------------------------------
	
		IF(velocity=0)THEN	
			state:=program_end;	
		END_IF	
		
	program_wait://-------------------------------------------------------------------------------------------
			
	program_end:
	
		finished:=TRUE;
		
	program_jog://-------------------------------------------------------------------------------------------
	
		IF(velocity=0 AND NOT jog_cmd.jog_enable)THEN	
			state:=program_end;	
		END_IF	
			
	program_error://-------------------------------------------------------------------------------------------
				
END_CASE

METHOD PRIVATE line_lenght : LREAL
VAR_INPUT
	p0,p1:sc_pnt;
END_VAR
line_lenght:=sqrt(expt(p1.x-p0.x,2)+expt(p1.y-p0.y,2)+expt(p1.z-p0.z,2));
END_METHOD

METHOD PRIVATE sc_char_is_letter : BOOL //return true if char on pos is letter
VAR_INPUT
	str : REFERENCE TO STRING(250);
	p:INT;
END_VAR
VAR
	pt : POINTER TO ARRAY[1..255] OF BYTE;
	X: BYTE;
END_VAR
pt := ADR(str);
X := pt^[p];

IF(X>64 AND X<91) THEN
	sc_char_is_letter:= TRUE;
ELSE
	sc_char_is_letter:= FALSE;
END_IF;
END_METHOD

METHOD PRIVATE sc_findp : int
VAR_INPUT
	str : STRING(250);
	src : STRING(250);
	p: INT;
END_VAR
VAR
	i: INT;
	ls: INT;
	lx: INT;
	stp: INT;
END_VAR
ls := LEN(str);
lx := LEN(src);
IF ls < lx OR lx = 0 THEN RETURN; END_IF;
stp := ls - lx + 1;
FOR i := MAX(p,1) TO stp DO
	IF MID(str,lx,i) = src THEN
		sc_findp := i;
		RETURN;
	END_IF;
END_FOR;
sc_findp := 0;
END_METHOD

METHOD PRIVATE sc_find_nonum : int
VAR_INPUT
	str : STRING(250);
	p : INT;
END_VAR
VAR
	i: INT;
	pt : POINTER TO ARRAY[1..255] OF BYTE;
	end: INT;
	X: BYTE;
END_VAR
pt := ADR(str);
end := LEN(str);
FOR i := MAX(p,1) TO end DO;
	X := pt^[i];
	IF (X < 48 AND X <> 46 AND X <> 45) OR X > 57 THEN
		sc_find_nonum := i;
		RETURN;
	END_IF;
END_FOR;
sc_find_nonum := 0;
END_METHOD

METHOD PRIVATE sc_find_num : int
VAR_INPUT
	str : STRING(250);
	p : INT;
END_VAR
VAR
	i : INT;
	pt : POINTER TO ARRAY[1..255] OF BYTE;
	stop : INT;
	X: BYTE;
END_VAR
pt := ADR(str);
stop := LEN(str);
FOR i := MAX(p,1) TO stop DO;
	X := pt^[i];
	IF (X > 47 AND X < 58) OR X = 46 OR X = 45 THEN
		sc_find_num := i;
		RETURN;
	END_IF;
END_FOR;
sc_find_num := 0;
END_METHOD

METHOD PRIVATE sc_get_letter : INT
VAR_INPUT
	str : REFERENCE TO STRING(250);//input string
	p : INT;//start position search value
	next_ptr:REFERENCE TO INT;//result line_pointer for next value search
END_VAR
VAR
	pt : POINTER TO ARRAY[1..255] OF BYTE;
	X: BYTE;
END_VAR
pt := ADR(str);
X := pt^[p];

IF(X>64 AND X<91) THEN
	sc_get_letter:=X;
ELSE
	sc_get_letter:=0;
END_IF;
next_ptr:=p+1;
END_METHOD

METHOD PRIVATE sc_get_value : LREAL
VAR_INPUT
	str : REFERENCE TO STRING(250);//input string
	p : INT;//start position search value
	next_ptr:REFERENCE TO INT;//result line_pointer for next letter search
END_VAR
VAR
	number_start: INT;
	letter_pos: INT;
	number_end: INT;
END_VAR
number_start:=sc_find_num(str,p);	
number_end:=sc_find_nonum(str,p);
IF(number_end=0)THEN
	number_end:=LEN(str)+1;
END_IF

sc_get_value:=STRING_TO_LREAL(MID(str,number_end-number_start,number_start));
//sc_get_value:=round(sc_get_value,DECIMALS);
next_ptr:=number_end;
END_METHOD

METHOD PRIVATE sc_parse_clean : BOOL
VAR_INPUT
END_VAR
//init parser last value, position tool ecc...
MEMUtils.MemSet(ADR(plv),0,SIZEOF(plv));
//init buffer 
parsed_vec.clear();

error_on_line:=0;	
syntax_error:=FALSE;
END_METHOD

METHOD PRIVATE sc_parse_line:UDINT
VAR_INPUT
	line:STRING(250);
END_VAR
VAR
	letter:ascii_letters;
	value:LREAL;
	char_ptr:INT;
	arc_radius:LREAL;
	p_block:sc_segment;// temp block for parsing
	
END_VAR
//init block
MEMUtils.MemSet(ADR(p_block),0,SIZEOF(p_block));

//uppercase
line:=uppercase(line);
//remove white space
line:=trim(line);

//start from 1 char of string
char_ptr:=1;
//check letter -> value
WHILE  sc_char_is_letter(line,char_ptr) DO		
	letter:=sc_get_letter(line,char_ptr,char_ptr);	
	CASE letter OF		
		G_:		
			value:=sc_get_value(line,char_ptr,char_ptr);			
			CASE LREAL_TO_INT(value) OF				
				0://rapid move
					p_block.primitive_id:=sc_primitive_id.rapid;		
				1://feed move
					p_block.primitive_id:=sc_primitive_id.line;		
				2://arc cw move
					p_block.primitive_id:=sc_primitive_id.arc_cw;
				3://arc ccw move
					p_block.primitive_id:=sc_primitive_id.arc_ccw;			
				4://dwell
								
				16://ijk plane
										
				17://xy plane
										
				18://zx plane
										
				19://yz plane
				
				43://tool compensation on

				49://tool compensation off
				
				90://absolute coord
					plv.abs_inc:=0;				
				91://relative coord
					plv.abs_inc:=1;
			END_CASE		
		X_:
			IF(plv.abs_inc=0)THEN				
				p_block.pnt_e.x:=sc_get_value(line,char_ptr,char_ptr);	
			ELSE
				p_block.pnt_e.x:=plv.pnt_e.x+sc_get_value(line,char_ptr,char_ptr);	
			END_IF									
		Y_:
			IF(plv.abs_inc=0)THEN				
				p_block.pnt_e.y:=sc_get_value(line,char_ptr,char_ptr);	
			ELSE
				p_block.pnt_e.y:=plv.pnt_e.y+sc_get_value(line,char_ptr,char_ptr);	
			END_IF																	
		Z_:
			IF(plv.abs_inc=0)THEN				
				p_block.pnt_e.z:=sc_get_value(line,char_ptr,char_ptr);	
			ELSE
				p_block.pnt_e.z:=plv.pnt_e.z+sc_get_value(line,char_ptr,char_ptr);	
			END_IF															
		A_:
			IF(plv.abs_inc=0)THEN				
				p_block.dir_e.a:=sc_get_value(line,char_ptr,char_ptr);	
			ELSE
				p_block.dir_e.a:=plv.dir_e.a+sc_get_value(line,char_ptr,char_ptr);	
			END_IF	
		B_:
			IF(plv.abs_inc=0)THEN				
				p_block.dir_e.b:=sc_get_value(line,char_ptr,char_ptr);	
			ELSE
				p_block.dir_e.b:=plv.dir_e.b+sc_get_value(line,char_ptr,char_ptr);	
			END_IF	
		C_:
			IF(plv.abs_inc=0)THEN				
				p_block.dir_e.c:=sc_get_value(line,char_ptr,char_ptr);	
			ELSE
				p_block.dir_e.c:=plv.dir_e.c+sc_get_value(line,char_ptr,char_ptr);	
			END_IF	
		U_:
			IF(plv.abs_inc=0)THEN				
				p_block.ext_e.u:=sc_get_value(line,char_ptr,char_ptr);	
			ELSE
				p_block.ext_e.u:=plv.ext_e.u+sc_get_value(line,char_ptr,char_ptr);	
			END_IF
		V_:
			IF(plv.abs_inc=0)THEN				
				p_block.ext_e.v:=sc_get_value(line,char_ptr,char_ptr);	
			ELSE
				p_block.ext_e.v:=plv.ext_e.v+sc_get_value(line,char_ptr,char_ptr);	
			END_IF
		W_:
			IF(plv.abs_inc=0)THEN				
				p_block.ext_e.w:=sc_get_value(line,char_ptr,char_ptr);	
			ELSE
				p_block.ext_e.w:=plv.ext_e.w+sc_get_value(line,char_ptr,char_ptr);	
			END_IF
		I_:
			p_block.pnt_c.x:=sc_get_value(line,char_ptr,char_ptr);		
		J_:
			p_block.pnt_c.y:=sc_get_value(line,char_ptr,char_ptr);	
		K_:
			p_block.pnt_c.z:=sc_get_value(line,char_ptr,char_ptr);	
		F_:
			plv.vel_max:=sc_get_value(line,char_ptr,char_ptr);	
		S_:
			plv.s_value:=LREAL_TO_UINT(sc_get_value(line,char_ptr,char_ptr));
		M_:
			value:=sc_get_value(line,char_ptr,char_ptr);			
			CASE LREAL_TO_INT(value) OF
				3://spindle cw
					plv.s_dir:=TRUE;
				4://spindle ccw
					plv.s_dir:=FALSE;
			END_CASE			
			p_block.m_value:=LREAL_TO_UINT(value);
		P_:
			p_block.p_value:=LREAL_TO_UINT(sc_get_value(line,char_ptr,char_ptr));
		T_:
			plv.t_value:=LREAL_TO_UINT(sc_get_value(line,char_ptr,char_ptr));
		H_:
			plv.h_value:=LREAL_TO_UINT(sc_get_value(line,char_ptr,char_ptr));
	END_CASE		
END_WHILE


//set start position from previous line end position
IF(p_block.primitive_id <> sc_primitive_id.empty)THEN
	
	IF(set_start_on_current_position)THEN
		set_start_on_current_position:=FALSE;		
		plv.pnt_s.x:=xyz.x;
		plv.pnt_s.y:=xyz.y;
		plv.pnt_s.z:=xyz.z;
	END_IF

	//update block start positions
	p_block.pnt_s:=plv.pnt_s;
	p_block.dir_s:=plv.dir_s;
	p_block.ext_s:=plv.ext_s;
	//line  
	IF(p_block.primitive_id=sc_primitive_id.line OR p_block.primitive_id=sc_primitive_id.rapid)THEN
		p_block.path_lenght:=line_lenght(p_block.pnt_s,p_block.pnt_e);
	//arc 
	ELSIF(p_block.primitive_id=sc_primitive_id.arc_ccw OR p_block.primitive_id=sc_primitive_id.arc_cw)THEN
		p_block.path_lenght:=arc_lenght(p_block.pnt_s,p_block.pnt_e,p_block.pnt_c,arc_radius);
		p_block.radius:=arc_radius;		
	END_IF
	//update last position on plv
	plv.pnt_s:=p_block.pnt_e;
	plv.dir_s:=p_block.dir_e;
	plv.ext_s:=p_block.ext_e;
ELSE
	p_block.pnt_s:=plv.pnt_s;
	p_block.dir_s:=plv.dir_s;
	p_block.ext_s:=plv.ext_s;
END_IF

p_block.traject_lenght_end:=p_block.path_lenght+plv.traject_lenght_end;
p_block.traject_lenght_begin:=p_block.traject_lenght_end-p_block.path_lenght;

//update trajectory lenght on plv
plv.traject_lenght_end:=p_block.traject_lenght_end;

//update block
IF(p_block.primitive_id=sc_primitive_id.rapid)THEN
	p_block.vel_max:=limits.max_vel;
ELSE
	p_block.vel_max:=plv.vel_max;
END_IF

IF(p_block.vel_max>limits.max_vel)THEN
	p_block.vel_max:=limits.max_vel;
END_IF
p_block.pnt_e:=plv.pnt_s;
p_block.dir_e:=plv.dir_s;
p_block.ext_e:=plv.ext_s;
p_block.s_value:=plv.s_value;
p_block.s_dir:=plv.s_dir;
p_block.t_value:=plv.t_value;
p_block.h_value:=plv.h_value;
p_block.gcode_line_nr:=plv.gcode_line_nr;
plv.gcode_line_nr:=plv.gcode_line_nr+1;

//add line to motion block buffer
parsed_vec.push_back(p_block);
END_METHOD

METHOD PRIVATE sc_parse_start : BOOL
VAR_INPUT
END_VAR
VAR
	i:UDINT;
	temp_line:STRING(250);
	comm_start:INT;
	comm_end:INT;
END_VAR
FOR i:=0 TO MAX_GCODE_LINE DO	
	//copy input string to temp
	temp_line:=gcode_lines[i];
	IF(temp_line='')THEN
		EXIT;
	END_IF;
	//find start comment <-
	comm_start:=sc_findp(temp_line,'(',1);
	IF(comm_start<>0)THEN
		i:=i+1;
		//jump comment line
		temp_line:=gcode_lines[i];
	END_IF	
	//parse line
	error_on_line:=sc_parse_line(temp_line);
	IF(UDINT_TO_BOOL(error_on_line))THEN
		syntax_error:=TRUE;
		EXIT;
	END_IF								
END_FOR
END_METHOD

METHOD PRIVATE to_upper : byte
VAR_INPUT
	IN : BYTE;
END_VAR
IF in > 96 AND in < 123 THEN
   TO_UPPER := in AND 16#DF;
ELSIF in > 223 AND in <> 247 AND in <> 255  THEN
   TO_UPPER := in AND 16#DF;
ELSE
   TO_UPPER := in;
END_IF;
END_METHOD

METHOD PRIVATE trim : string
VAR_INPUT
	str : STRING(250);
END_VAR
VAR
	p: INT;
END_VAR
TRIM := str;
REPEAT
	p := FIND(trim,' ');
	IF p > 0 THEN TRIM := REPLACE(TRIM,'',1,p); END_IF;
UNTIL p = 0	END_REPEAT;
END_METHOD

METHOD PRIVATE uppercase : STRING
VAR_INPUT
	str : STRING(250);
END_VAR
VAR
	pt : POINTER TO BYTE;
	p: INT;
	l: INT;
END_VAR
pt := ADR(UPPERCASE);
UPPERCASE := str;
l := LEN(str);
FOR p := 1 TO l DO
	pt^ := TO_UPPER(pt^);
	pt := pt + 1;
END_FOR;
END_METHOD

METHOD PRIVATE arc_lenght : LREAL
VAR_INPUT
	p1:sc_pnt;//! start position
	p2:sc_pnt;//! end position 
	center:sc_pnt;//! center IJK
	arc_radius:REFERENCE TO LREAL;//! radius result
END_VAR
VAR
	radius:LREAL;
	circumference:LREAL;
	startingAngle,endingAngle:LREAL;
	chordSquared,tau,chordHeight:LREAL;
	theta:LREAL;
END_VAR
// add center offset IJ
center.x:=center.x+p1.x;
center.y:=center.y+p1.y;
// Compute geometry.
radius:=SQRT(EXPT(center.x-p1.x,2)+EXPT(center.y-p1.y,2)); 
circumference:=2.0*M_PI*radius;
startingAngle:=math.atan2(p1.y-center.y,p1.x-center.x);
endingAngle:=math.atan2(p2.y-center.y,p2.x-center.x);

// Compute chord height of arc.
chordSquared:=SQRT(EXPT(p2.x-p1.x,2)+EXPT(p2.y-p1.y,2));
tau:= (EXPT(radius,2)-(chordSquared/4));
chordHeight := radius - tau;

// Compute angle between lines.
theta:=endingAngle-startingAngle;
	//COUNTERCLOCKWISE
	IF (theta < 0)THEN
		theta:=theta+2*M_PI;
	END_IF
 
	//CLOCKWISE
	IF (theta >= 0)THEN	
		theta:=theta-2*M_PI;;
	END_IF


arc_lenght:=ABS(circumference*(theta/(2*M_PI)));
arc_radius:=radius;
END_METHOD

METHOD line_arc_angle : bool
VAR_INPUT
	p0:sc_pnt;
	p1:sc_pnt;
	p2:sc_pnt;
	p3:sc_pnt;
	angle_deg:REFERENCE TO LREAL;
END_VAR
VAR
	pi:sc_pnt;
END_VAR
interpolate_arc(p1,p2,p3,0.1,pi);
line_line_angle(p0,p1,pi,angle_deg);
END_METHOD

METHOD arc_arc_angle : bool
VAR_INPUT
	p0:sc_pnt;
	p1:sc_pnt;
	p2:sc_pnt;
	p3:sc_pnt;
	p4:sc_pnt;
	angle_deg:REFERENCE TO LREAL;
END_VAR
VAR
	pi0,pi1:sc_pnt;
	
END_VAR
interpolate_arc(p0,p1,p2,0.9,pi0);
interpolate_arc(p2,p3,p4,0.1,pi1);
line_line_angle(pi0,p2,pi1,angle_deg);
END_METHOD

